LIN {X 0,Y 573.283,Z 236.698,A -85,B 0,C 180,E1 -2312.234,E2 -2312.234} C_VEL
LIN {X 0,Y 573.268,Z 236.699,A -85,B 0,C 180,E1 -2315.365,E2 -2315.365} C_VEL
LIN {X 0,Y 573.222,Z 236.703,A -85,B 0,C 180,E1 -2318.418,E2 -2318.418} C_VEL
LIN {X 0,Y 573.27,Z 236.695,A -85,B 0,C 180,E1 -2320.727,E2 -2320.727} C_VEL
LIN {X 0,Y 573.253,Z 236.706,A -85,B 0,C 180,E1 -2323.621,E2 -2323.621} C_VEL
LIN {X 0,Y 573.232,Z 236.7,A -85,B 0,C 180,E1 -2326.529,E2 -2326.529} C_VEL
LIN {X 0,Y 573.274,Z 236.694,A -85,B 0,C 180,E1 -2328.733,E2 -2328.733} C_VEL
LIN {X 0,Y 573.298,Z 236.7,A -85,B 0,C 180,E1 -2331.54,E2 -2331.54} C_VEL
LIN {X 0,Y 573.285,Z 236.694,A -85,B 0,C 180,E1 -2334.371,E2 -2334.371} C_VEL
LIN {X 0,Y 573.304,Z 236.698,A -85,B 0,C 180,E1 -2337.188,E2 -2337.188} C_VEL
LIN {X 0,Y 573.307,Z 236.691,A -85,B 0,C 180,E1 -2339.999,E2 -2339.999} C_VEL
LIN {X 0,Y 573.305,Z 236.694,A -85,B 0,C 180,E1 -2342.81,E2 -2342.81} C_VEL
LIN {X 0,Y 573.282,Z 236.696,A -85,B 0,C 180,E1 -2345.627,E2 -2345.627} C_VEL
LIN {X 0,Y 573.279,Z 236.696,A -85,B 0,C 180,E1 -2348.458,E2 -2348.458} C_VEL
LIN {X 0,Y 573.287,Z 236.699,A -85,B 0,C 180,E1 -2351.311,E2 -2351.311} C_VEL
LIN {X 0,Y 573.268,Z 236.697,A -85,B 0,C 180,E1 -2354.424,E2 -2354.424} C_VEL
LIN {X 0,Y 573.246,Z 236.705,A -85,B 0,C 180,E1 -2357.111,E2 -2357.111} C_VEL
LIN {X 0,Y 573.245,Z 236.699,A -85,B 0,C 180,E1 -2360.076,E2 -2360.076} C_VEL
LIN {X 0,Y 573.258,Z 236.7,A -85,B 0,C 180,E1 -2363.153,E2 -2363.153} C_VEL
LIN {X 0,Y 573.241,Z 236.703,A -85,B 0,C 180,E1 -2364.403,E2 -2364.403} C_VEL
LIN {X 0,Y 572.608,Z 236.788,A -85,B 0,C 180,E1 -2364.99,E2 -2364.99} C_VEL
LIN {X 0,Y 569.762,Z 237.142,A -85,B 0,C 180,E1 -2365.941,E2 -2365.941} C_VEL
LIN {X 0,Y 567.334,Z 237.444,A -85,B 0,C 180,E1 -2366.707,E2 -2366.707} C_VEL
LIN {X 0,Y 566.285,Z 237.568,A -85,B 0,C 180,E1 -2367.298,E2 -2367.298} C_VEL
LIN {X 0,Y 566.197,Z 237.577,A -85,B 0,C 180,E1 -2367.498,E2 -2367.498} C_VEL
LIN {X 0,Y 566.212,Z 237.574,A -85,B 0,C 180,E1 -2369.767,E2 -2369.767} C_VEL
LIN {X 0,Y 566.191,Z 237.584,A -85,B 0,C 180,E1 -2372.43,E2 -2372.43} C_VEL
LIN {X 0,Y 566.188,Z 237.579,A -85,B 0,C 180,E1 -2374.992,E2 -2374.992} C_VEL
LIN {X 0,Y 566.181,Z 237.579,A -85,B 0,C 180,E1 -2377.46,E2 -2377.46} C_VEL
LIN {X 0,Y 566.212,Z 237.581,A -85,B 0,C 180,E1 -2380.197,E2 -2380.197} C_VEL
LIN {X 0,Y 566.196,Z 237.578,A -85,B 0,C 180,E1 -2383.053,E2 -2383.053} C_VEL
LIN {X 0,Y 566.186,Z 237.585,A -85,B 0,C 180,E1 -2386.048,E2 -2386.048} C_VEL
LIN {X 0,Y 566.196,Z 237.579,A -85,B 0,C 180,E1 -2388.864,E2 -2388.864} C_VEL
LIN {X 0,Y 566.175,Z 237.584,A -85,B 0,C 180,E1 -2391.637,E2 -2391.637} C_VEL
LIN {X 0,Y 566.214,Z 237.686,A -85,B 0,C 180,E1 -2394.485,E2 -2394.485} C_VEL
LIN {X 0,Y 566.846,Z 243.491,A -85,B 0,C 180,E1 -2395.444,E2 -2395.444} C_VEL
LIN {X 0,Y 566.584,Z 259.614,A -85,B 0,C 180,E1 -2397.977,E2 -2397.977} C_VEL
LIN {X 0,Y 566.546,Z 266.895,A -85,B 0,C 180,E1 -2399.084,E2 -2399.084} C_VEL
LIN {X 0,Y 567.77,Z 274.286,A -85,B 0,C 180,E1 -2399.217,E2 -2399.217} C_VEL
LIN {X 0,Y 567.426,Z 403.279,A -85,B 0,C 180,E1 -2400.888,E2 -2400.888} C_VEL
LIN {X 0,Y 567.276,Z 417.794,A -85,B 0,C 180,E1 -2401.223,E2 -2401.223} C_VEL
LIN {X 0,Y 567.143,Z 431.004,A -85,B 0,C 180,E1 -2401.667,E2 -2401.667} C_VEL
LIN {X 0,Y 566.989,Z 443.123,A -85,B 0,C 180,E1 -2402.202,E2 -2402.202} C_VEL
LIN {X 0,Y 566.761,Z 456.118,A -85,B 0,C 180,E1 -2402.929,E2 -2402.929} C_VEL
LIN {X 0,Y 566.557,Z 468.236,A -85,B 0,C 180,E1 -2403.774,E2 -2403.774} C_VEL
LIN {X 0,Y 566.389,Z 479.468,A -85,B 0,C 180,E1 -2404.731,E2 -2404.731} C_VEL
LIN {X 0,Y 566.253,Z 490.014,A -85,B 0,C 180,E1 -2405.822,E2 -2405.822} C_VEL
LIN {X 0,Y 566.139,Z 499.355,A -85,B 0,C 180,E1 -2406.999,E2 -2406.999} C_VEL
LIN {X 0,Y 566.041,Z 506.752,A -85,B 0,C 180,E1 -2408.132,E2 -2408.132} C_VEL
LIN {X 0,Y 565.961,Z 512.883,A -85,B 0,C 180,E1 -2409.274,E2 -2409.274} C_VEL
LIN {X 0,Y 565.955,Z 518.916,A -85,B 0,C 180,E1 -2410.688,E2 -2410.688} C_VEL
LIN {X 0,Y 565.898,Z 522.863,A -85,B 0,C 180,E1 -2411.912,E2 -2411.912} C_VEL
LIN {X 0,Y 565.861,Z 526.209,A -85,B 0,C 180,E1 -2413.402,E2 -2413.402} C_VEL
LIN {X 0,Y 565.827,Z 528.034,A -85,B 0,C 180,E1 -2414.881,E2 -2414.881} C_VEL
LIN {X 0,Y 565.854,Z 528.439,A -85,B 0,C 180,E1 -2416.351,E2 -2416.351} C_VEL
LIN {X 0,Y 565.859,Z 527.454,A -85,B 0,C 180,E1 -2417.811,E2 -2417.811} C_VEL
LIN {X 0,Y 565.879,Z 525.08,A -85,B 0,C 180,E1 -2419.264,E2 -2419.264} C_VEL
LIN {X 0,Y 565.878,Z 521.281,A -85,B 0,C 180,E1 -2420.709,E2 -2420.709} C_VEL
LIN {X 0,Y 565.952,Z 517.395,A -85,B 0,C 180,E1 -2421.79,E2 -2421.79} C_VEL
LIN {X 0,Y 565.985,Z 511.373,A -85,B 0,C 180,E1 -2423.115,E2 -2423.115} C_VEL
LIN {X 0,Y 566.037,Z 504.637,A -85,B 0,C 180,E1 -2424.3,E2 -2424.3} C_VEL
LIN {X 0,Y 566.174,Z 495.909,A -85,B 0,C 180,E1 -2425.551,E2 -2425.551} C_VEL
LIN {X 0,Y 566.285,Z 486.831,A -85,B 0,C 180,E1 -2426.621,E2 -2426.621} C_VEL
LIN {X 0,Y 566.438,Z 477.817,A -85,B 0,C 180,E1 -2427.511,E2 -2427.511} C_VEL
LIN {X 0,Y 566.611,Z 465.974,A -85,B 0,C 180,E1 -2428.49,E2 -2428.49} C_VEL
LIN {X 0,Y 566.825,Z 454.056,A -85,B 0,C 180,E1 -2429.29,E2 -2429.29} C_VEL
LIN {X 0,Y 567.036,Z 440.812,A -85,B 0,C 180,E1 -2430,E2 -2430} C_VEL
LIN {X 0,Y 567.188,Z 426.85,A -85,B 0,C 180,E1 -2430.577,E2 -2430.577} C_VEL
LIN {X 0,Y 567.32,Z 412.804,A -85,B 0,C 180,E1 -2430.998,E2 -2430.998} C_VEL
LIN {X 0,Y 567.413,Z 399.298,A -85,B 0,C 180,E1 -2431.264,E2 -2431.264} C_VEL
LIN {X 0,Y 567.674,Z 272.851,A -85,B 0,C 180,E1 -2432.894,E2 -2432.894} C_VEL
LIN {X 0,Y 566.499,Z 266.67,A -85,B 0,C 180,E1 -2433.022,E2 -2433.022} C_VEL
LIN {X 0,Y 566.729,Z 250.62,A -85,B 0,C 180,E1 -2435.515,E2 -2435.515} C_VEL
LIN {X 0,Y 566.793,Z 240.515,A -85,B 0,C 180,E1 -2437.123,E2 -2437.123} C_VEL
LIN {X 0,Y 566.242,Z 237.58,A -85,B 0,C 180,E1 -2437.65,E2 -2437.65} C_VEL
LIN {X 0,Y 566.238,Z 237.573,A -85,B 0,C 180,E1 -2440.73,E2 -2440.73} C_VEL
LIN {X 0,Y 566.194,Z 237.584,A -85,B 0,C 180,E1 -2443.641,E2 -2443.641} C_VEL
LIN {X 0,Y 566.21,Z 237.575,A -85,B 0,C 180,E1 -2446.588,E2 -2446.588} C_VEL
LIN {X 0,Y 566.201,Z 237.582,A -85,B 0,C 180,E1 -2449.581,E2 -2449.581} C_VEL
LIN {X 0,Y 566.184,Z 237.586,A -85,B 0,C 180,E1 -2451.863,E2 -2451.863} C_VEL
LIN {X 0,Y 566.22,Z 237.575,A -85,B 0,C 180,E1 -2455.034,E2 -2455.034} C_VEL
LIN {X 0,Y 566.214,Z 237.579,A -85,B 0,C 180,E1 -2457.338,E2 -2457.338} C_VEL
LIN {X 0,Y 566.214,Z 237.581,A -85,B 0,C 180,E1 -2459.767,E2 -2459.767} C_VEL
LIN {X 0,Y 566.198,Z 237.576,A -85,B 0,C 180,E1 -2462.432,E2 -2462.432} C_VEL
LIN {X 0,Y 566.201,Z 237.578,A -85,B 0,C 180,E1 -2464.995,E2 -2464.995} C_VEL
LIN {X 0,Y 566.183,Z 237.588,A -85,B 0,C 180,E1 -2467.461,E2 -2467.461} C_VEL
LIN {X 0,Y 566.213,Z 237.575,A -85,B 0,C 180,E1 -2470.198,E2 -2470.198} C_VEL
LIN {X 0,Y 566.198,Z 237.581,A -85,B 0,C 180,E1 -2473.053,E2 -2473.053} C_VEL
LIN {X 0,Y 566.188,Z 237.578,A -85,B 0,C 180,E1 -2476.049,E2 -2476.049} C_VEL
LIN {X 0,Y 566.207,Z 237.579,A -85,B 0,C 180,E1 -2478.865,E2 -2478.865} C_VEL
LIN {X 0,Y 566.179,Z 237.582,A -85,B 0,C 180,E1 -2481.638,E2 -2481.638} C_VEL
LIN {X 0,Y 566.2,Z 237.576,A -85,B 0,C 180,E1 -2484.312,E2 -2484.312} C_VEL
LIN {X 0,Y 566.215,Z 237.581,A -85,B 0,C 180,E1 -2486.899,E2 -2486.899} C_VEL
LIN {X 0,Y 566.182,Z 237.582,A -85,B 0,C 180,E1 -2489.409,E2 -2489.409} C_VEL
LIN {X 0,Y 566.215,Z 237.574,A -85,B 0,C 180,E1 -2491.859,E2 -2491.859} C_VEL
LIN {X 0,Y 566.214,Z 237.575,A -85,B 0,C 180,E1 -2494.252,E2 -2494.252} C_VEL
LIN {X 0,Y 566.181,Z 237.585,A -85,B 0,C 180,E1 -2496.714,E2 -2496.714} C_VEL
LIN {X 0,Y 566.209,Z 237.575,A -85,B 0,C 180,E1 -2499.664,E2 -2499.664} C_VEL
LIN {X 0,Y 566.194,Z 237.584,A -85,B 0,C 180,E1 -2502.669,E2 -2502.669} C_VEL
LIN {X 0,Y 566.223,Z 237.573,A -85,B 0,C 180,E1 -2505.628,E2 -2505.628} C_VEL
LIN {X 0,Y 566.223,Z 237.583,A -85,B 0,C 180,E1 -2508.676,E2 -2508.676} C_VEL
LIN {X 0,Y 566.226,Z 237.573,A -85,B 0,C 180,E1 -2511.435,E2 -2511.435} C_VEL
LIN {X 0,Y 566.253,Z 237.575,A -85,B 0,C 180,E1 -2514.303,E2 -2514.303} C_VEL
LIN {X 0,Y 566.272,Z 237.568,A -85,B 0,C 180,E1 -2517.867,E2 -2517.867} C_VEL
LIN {X 0,Y 566.298,Z 237.57,A -85,B 0,C 180,E1 -2520.712,E2 -2520.712} C_VEL
LIN {X 0,Y 566.269,Z 237.571,A -85,B 0,C 180,E1 -2522.846,E2 -2522.846} C_VEL
LIN {X 0,Y 566.254,Z 237.57,A -85,B 0,C 180,E1 -2525.699,E2 -2525.699} C_VEL
LIN {X 0,Y 566.227,Z 237.579,A -85,B 0,C 180,E1 -2528.567,E2 -2528.567} C_VEL
LIN {X 0,Y 566.234,Z 237.572,A -85,B 0,C 180,E1 -2531.455,E2 -2531.455} C_VEL
LIN {X 0,Y 566.227,Z 237.578,A -85,B 0,C 180,E1 -2534.508,E2 -2534.508} C_VEL
LIN {X 0,Y 566.198,Z 237.577,A -85,B 0,C 180,E1 -2537.332,E2 -2537.332} C_VEL
LIN {X 0,Y 566.209,Z 237.581,A -85,B 0,C 180,E1 -2540.338,E2 -2540.338} C_VEL
LIN {X 0,Y 566.185,Z 237.579,A -85,B 0,C 180,E1 -2543.405,E2 -2543.405} C_VEL
LIN {X 0,Y 566.209,Z 237.58,A -85,B 0,C 180,E1 -2545.75,E2 -2545.75} C_VEL
LIN {X 0,Y 566.201,Z 237.582,A -85,B 0,C 180,E1 -2548.204,E2 -2548.204} C_VEL
LIN {X 0,Y 566.189,Z 237.578,A -85,B 0,C 180,E1 -2550.593,E2 -2550.593} C_VEL
LIN {X 0,Y 566.225,Z 237.573,A -85,B 0,C 180,E1 -2553.103,E2 -2553.103} C_VEL
LIN {X 0,Y 566.209,Z 237.582,A -85,B 0,C 180,E1 -2555.689,E2 -2555.689} C_VEL
LIN {X 0,Y 566.213,Z 237.575,A -85,B 0,C 180,E1 -2558.56,E2 -2558.56} C_VEL
LIN {X 0,Y 566.201,Z 237.578,A -85,B 0,C 180,E1 -2561.138,E2 -2561.138} C_VEL
LIN {X 0,Y 566.195,Z 237.581,A -85,B 0,C 180,E1 -2564.037,E2 -2564.037} C_VEL
LIN {X 0,Y 566.204,Z 237.578,A -85,B 0,C 180,E1 -2567.083,E2 -2567.083} C_VEL
LIN {X 0,Y 566.205,Z 237.582,A -85,B 0,C 180,E1 -2569.802,E2 -2569.802} C_VEL
LIN {X 0,Y 566.197,Z 237.576,A -85,B 0,C 180,E1 -2572.6,E2 -2572.6} C_VEL
LIN {X 0,Y 566.199,Z 237.581,A -85,B 0,C 180,E1 -2575.182,E2 -2575.182} C_VEL
LIN {X 0,Y 566.233,Z 237.579,A -85,B 0,C 180,E1 -2577.744,E2 -2577.744} C_VEL
LIN {X 0,Y 566.203,Z 237.577,A -85,B 0,C 180,E1 -2580.329,E2 -2580.329} C_VEL
LIN {X 0,Y 566.212,Z 237.578,A -85,B 0,C 180,E1 -2582.662,E2 -2582.662} C_VEL
LIN {X 0,Y 566.263,Z 237.689,A -85,B 0,C 180,E1 -2585.261,E2 -2585.261} C_VEL
LIN {X 0,Y 567.317,Z 243.08,A -85,B 0,C 180,E1 -2586.044,E2 -2586.044} C_VEL
LIN {X 0,Y 567.119,Z 262.492,A -85,B 0,C 180,E1 -2588.647,E2 -2588.647} C_VEL
LIN {X 0,Y 566.829,Z 284.536,A -85,B 0,C 180,E1 -2591.569,E2 -2591.569} C_VEL
LIN {X 0,Y 566.669,Z 295.557,A -85,B 0,C 180,E1 -2593.018,E2 -2593.018} C_VEL
LIN {X 0,Y 567.791,Z 302.851,A -85,B 0,C 180,E1 -2593.155,E2 -2593.155} C_VEL
LIN {X 0,Y 567.434,Z 433.897,A -85,B 0,C 180,E1 -2594.856,E2 -2594.856} C_VEL
LIN {X 0,Y 567.268,Z 448.613,A -85,B 0,C 180,E1 -2595.202,E2 -2595.202} C_VEL
LIN {X 0,Y 567.112,Z 462.843,A -85,B 0,C 180,E1 -2595.696,E2 -2595.696} C_VEL
LIN {X 0,Y 566.963,Z 475.645,A -85,B 0,C 180,E1 -2596.286,E2 -2596.286} C_VEL
LIN {X 0,Y 566.755,Z 488.106,A -85,B 0,C 180,E1 -2597.012,E2 -2597.012} C_VEL
LIN {X 0,Y 566.572,Z 500.647,A -85,B 0,C 180,E1 -2597.917,E2 -2597.917} C_VEL
LIN {X 0,Y 566.447,Z 511.321,A -85,B 0,C 180,E1 -2598.861,E2 -2598.861} C_VEL
LIN {X 0,Y 566.206,Z 521.853,A -85,B 0,C 180,E1 -2599.993,E2 -2599.993} C_VEL
LIN {X 0,Y 566.137,Z 530.174,A -85,B 0,C 180,E1 -2601.073,E2 -2601.073} C_VEL
LIN {X 0,Y 566.047,Z 538.128,A -85,B 0,C 180,E1 -2602.33,E2 -2602.33} C_VEL
LIN {X 0,Y 565.945,Z 544.528,A -85,B 0,C 180,E1 -2603.583,E2 -2603.583} C_VEL
LIN {X 0,Y 565.928,Z 548.961,A -85,B 0,C 180,E1 -2604.656,E2 -2604.656} C_VEL
LIN {X 0,Y 565.956,Z 552.443,A -85,B 0,C 180,E1 -2605.727,E2 -2605.727} C_VEL
LIN {X 0,Y 565.875,Z 555.832,A -85,B 0,C 180,E1 -2607.152,E2 -2607.152} C_VEL
LIN {X 0,Y 565.841,Z 557.833,A -85,B 0,C 180,E1 -2608.577,E2 -2608.577} C_VEL
LIN {X 0,Y 565.837,Z 558.5,A -85,B 0,C 180,E1 -2610,E2 -2610} C_VEL
LIN {X 0,Y 565.841,Z 557.834,A -85,B 0,C 180,E1 -2611.423,E2 -2611.423} C_VEL
LIN {X 0,Y 565.875,Z 555.835,A -85,B 0,C 180,E1 -2612.847,E2 -2612.847} C_VEL
LIN {X 0,Y 565.956,Z 552.446,A -85,B 0,C 180,E1 -2614.273,E2 -2614.273} C_VEL
LIN {X 0,Y 565.985,Z 547.569,A -85,B 0,C 180,E1 -2615.701,E2 -2615.701} C_VEL
LIN {X 0,Y 565.996,Z 543.045,A -85,B 0,C 180,E1 -2616.738,E2 -2616.738} C_VEL
LIN {X 0,Y 566.047,Z 536.038,A -85,B 0,C 180,E1 -2618.029,E2 -2618.029} C_VEL
LIN {X 0,Y 566.177,Z 527.56,A -85,B 0,C 180,E1 -2619.286,E2 -2619.286} C_VEL
LIN {X 0,Y 566.294,Z 518.71,A -85,B 0,C 180,E1 -2620.367,E2 -2620.367} C_VEL
LIN {X 0,Y 566.467,Z 507.992,A -85,B 0,C 180,E1 -2621.449,E2 -2621.449} C_VEL
LIN {X 0,Y 566.611,Z 497.143,A -85,B 0,C 180,E1 -2622.354,E2 -2622.354} C_VEL
LIN {X 0,Y 566.79,Z 485.26,A -85,B 0,C 180,E1 -2623.17,E2 -2623.17} C_VEL
LIN {X 0,Y 567.035,Z 472.104,A -85,B 0,C 180,E1 -2623.894,E2 -2623.894} C_VEL
LIN {X 0,Y 567.235,Z 459.039,A -85,B 0,C 180,E1 -2624.453,E2 -2624.453} C_VEL
LIN {X 0,Y 567.354,Z 445.151,A -85,B 0,C 180,E1 -2624.893,E2 -2624.893} C_VEL
LIN {X 0,Y 567.428,Z 431.157,A -85,B 0,C 180,E1 -2625.19,E2 -2625.19} C_VEL
LIN {X 0,Y 567.737,Z 301.687,A -85,B 0,C 180,E1 -2626.862,E2 -2626.862} C_VEL
LIN {X 0,Y 566.666,Z 295.559,A -85,B 0,C 180,E1 -2626.982,E2 -2626.982} C_VEL
LIN {X 0,Y 566.964,Z 274.789,A -85,B 0,C 180,E1 -2629.722,E2 -2629.722} C_VEL
LIN {X 0,Y 567.271,Z 253.229,A -85,B 0,C 180,E1 -2632.585,E2 -2632.585} C_VEL
LIN {X 0,Y 567.297,Z 243.048,A -85,B 0,C 180,E1 -2633.958,E2 -2633.958} C_VEL
LIN {X 0,Y 566.256,Z 237.58,A -85,B 0,C 180,E1 -2634.763,E2 -2634.763} C_VEL
LIN {X 0,Y 566.211,Z 237.577,A -85,B 0,C 180,E1 -2637.338,E2 -2637.338} C_VEL
LIN {X 0,Y 566.201,Z 237.578,A -85,B 0,C 180,E1 -2639.768,E2 -2639.768} C_VEL
LIN {X 0,Y 566.206,Z 237.585,A -85,B 0,C 180,E1 -2642.43,E2 -2642.43} C_VEL
LIN {X 0,Y 566.18,Z 237.583,A -85,B 0,C 180,E1 -2644.989,E2 -2644.989} C_VEL
LIN {X 0,Y 566.194,Z 237.577,A -85,B 0,C 180,E1 -2647.46,E2 -2647.46} C_VEL
LIN {X 0,Y 566.204,Z 237.584,A -85,B 0,C 180,E1 -2650.198,E2 -2650.198} C_VEL
LIN {X 0,Y 566.203,Z 237.577,A -85,B 0,C 180,E1 -2653.053,E2 -2653.053} C_VEL
LIN {X 0,Y 566.195,Z 237.584,A -85,B 0,C 180,E1 -2656.048,E2 -2656.048} C_VEL
LIN {X 0,Y 566.208,Z 237.577,A -85,B 0,C 180,E1 -2658.863,E2 -2658.863} C_VEL
LIN {X 0,Y 566.186,Z 237.581,A -85,B 0,C 180,E1 -2661.636,E2 -2661.636} C_VEL
LIN {X 0,Y 566.208,Z 237.578,A -85,B 0,C 180,E1 -2664.311,E2 -2664.311} C_VEL
LIN {X 0,Y 566.224,Z 237.574,A -85,B 0,C 180,E1 -2666.897,E2 -2666.897} C_VEL
LIN {X 0,Y 566.188,Z 237.579,A -85,B 0,C 180,E1 -2669.407,E2 -2669.407} C_VEL
LIN {X 0,Y 566.222,Z 237.582,A -85,B 0,C 180,E1 -2671.857,E2 -2671.857} C_VEL
LIN {X 0,Y 566.208,Z 237.579,A -85,B 0,C 180,E1 -2674.25,E2 -2674.25} C_VEL
LIN {X 0,Y 566.185,Z 237.578,A -85,B 0,C 180,E1 -2676.713,E2 -2676.713} C_VEL
LIN {X 0,Y 566.208,Z 237.584,A -85,B 0,C 180,E1 -2679.662,E2 -2679.662} C_VEL
LIN {X 0,Y 566.197,Z 237.577,A -85,B 0,C 180,E1 -2682.668,E2 -2682.668} C_VEL
LIN {X 0,Y 566.226,Z 237.583,A -85,B 0,C 180,E1 -2685.626,E2 -2685.626} C_VEL
LIN {X 0,Y 566.267,Z 237.567,A -85,B 0,C 180,E1 -2688.653,E2 -2688.653} C_VEL
LIN {X 0,Y 566.24,Z 237.581,A -85,B 0,C 180,E1 -2691.434,E2 -2691.434} C_VEL
LIN {X 0,Y 566.252,Z 237.57,A -85,B 0,C 180,E1 -2694.301,E2 -2694.301} C_VEL
LIN {X 0,Y 566.27,Z 237.574,A -85,B 0,C 180,E1 -2697.154,E2 -2697.154} C_VEL
LIN {X 0,Y 566.277,Z 237.567,A -85,B 0,C 180,E1 -2699.999,E2 -2699.999} C_VEL
LIN {X 0,Y 566.27,Z 237.571,A -85,B 0,C 180,E1 -2702.845,E2 -2702.845} C_VEL
LIN {X 0,Y 566.25,Z 237.571,A -85,B 0,C 180,E1 -2705.697,E2 -2705.697} C_VEL
LIN {X 0,Y 566.223,Z 237.576,A -85,B 0,C 180,E1 -2708.565,E2 -2708.565} C_VEL
LIN {X 0,Y 566.239,Z 237.575,A -85,B 0,C 180,E1 -2711.453,E2 -2711.453} C_VEL
LIN {X 0,Y 566.221,Z 237.576,A -85,B 0,C 180,E1 -2714.506,E2 -2714.506} C_VEL
LIN {X 0,Y 566.188,Z 237.581,A -85,B 0,C 180,E1 -2717.331,E2 -2717.331} C_VEL
LIN {X 0,Y 566.208,Z 237.578,A -85,B 0,C 180,E1 -2720.336,E2 -2720.336} C_VEL
LIN {X 0,Y 566.217,Z 237.575,A -85,B 0,C 180,E1 -2723.401,E2 -2723.401} C_VEL
LIN {X 0,Y 566.199,Z 237.577,A -85,B 0,C 180,E1 -2725.748,E2 -2725.748} C_VEL
LIN {X 0,Y 566.197,Z 237.577,A -85,B 0,C 180,E1 -2727.498,E2 -2727.498} C_VEL
LIN {X 0,Y 565.523,Z 237.664,A -85,B 0,C 180,E1 -2728.092,E2 -2728.092} C_VEL
LIN {X 0,Y 562.659,Z 238.02,A -85,B 0,C 180,E1 -2729.055,E2 -2729.055} C_VEL
LIN {X 0,Y 560.246,Z 238.32,A -85,B 0,C 180,E1 -2729.831,E2 -2729.831} C_VEL
LIN {X 0,Y 559.214,Z 238.452,A -85,B 0,C 180,E1 -2730.43,E2 -2730.43} C_VEL
LIN {X 0,Y 559.133,Z 238.457,A -85,B 0,C 180,E1 -2730.633,E2 -2730.633} C_VEL
LIN {X 0,Y 559.149,Z 238.455,A -85,B 0,C 180,E1 -2733.574,E2 -2733.574} C_VEL
LIN {X 0,Y 559.152,Z 238.462,A -85,B 0,C 180,E1 -2736.448,E2 -2736.448} C_VEL
LIN {X 0,Y 559.163,Z 238.455,A -85,B 0,C 180,E1 -2738.933,E2 -2738.933} C_VEL
LIN {X 0,Y 559.18,Z 238.453,A -85,B 0,C 180,E1 -2741.767,E2 -2741.767} C_VEL
LIN {X 0,Y 559.124,Z 238.462,A -85,B 0,C 180,E1 -2744.739,E2 -2744.739} C_VEL
LIN {X 0,Y 559.148,Z 238.456,A -85,B 0,C 180,E1 -2747.257,E2 -2747.257} C_VEL
LIN {X 0,Y 559.171,Z 238.462,A -85,B 0,C 180,E1 -2750.135,E2 -2750.135} C_VEL
LIN {X 0,Y 559.13,Z 238.462,A -85,B 0,C 180,E1 -2752.892,E2 -2752.892} C_VEL
LIN {X 0,Y 559.207,Z 238.602,A -85,B 0,C 180,E1 -2754.323,E2 -2754.323} C_VEL
LIN {X 0,Y 559.951,Z 243.649,A -85,B 0,C 180,E1 -2755.176,E2 -2755.176} C_VEL
LIN {X 0,Y 559.606,Z 261.03,A -85,B 0,C 180,E1 -2757.954,E2 -2757.954} C_VEL
LIN {X 0,Y 559.567,Z 266.769,A -85,B 0,C 180,E1 -2758.864,E2 -2758.864} C_VEL
LIN {X 0,Y 560.963,Z 274.225,A -85,B 0,C 180,E1 -2759.006,E2 -2759.006} C_VEL
LIN {X 0,Y 560.582,Z 403.558,A -85,B 0,C 180,E1 -2760.704,E2 -2760.704} C_VEL
LIN {X 0,Y 560.409,Z 417.899,A -85,B 0,C 180,E1 -2761.04,E2 -2761.04} C_VEL
LIN {X 0,Y 560.236,Z 432.09,A -85,B 0,C 180,E1 -2761.531,E2 -2761.531} C_VEL
LIN {X 0,Y 560.033,Z 445.125,A -85,B 0,C 180,E1 -2762.131,E2 -2762.131} C_VEL
LIN {X 0,Y 559.806,Z 457.281,A -85,B 0,C 180,E1 -2762.839,E2 -2762.839} C_VEL
LIN {X 0,Y 559.566,Z 469.557,A -85,B 0,C 180,E1 -2763.723,E2 -2763.723} C_VEL
LIN {X 0,Y 559.384,Z 480.79,A -85,B 0,C 180,E1 -2764.713,E2 -2764.713} C_VEL
LIN {X 0,Y 559.214,Z 490.045,A -85,B 0,C 180,E1 -2765.696,E2 -2765.696} C_VEL
LIN {X 0,Y 559.105,Z 498.891,A -85,B 0,C 180,E1 -2766.82,E2 -2766.82} C_VEL
LIN {X 0,Y 558.963,Z 506.712,A -85,B 0,C 180,E1 -2768.024,E2 -2768.024} C_VEL
LIN {X 0,Y 558.906,Z 511.946,A -85,B 0,C 180,E1 -2769,E2 -2769} C_VEL
LIN {X 0,Y 558.865,Z 517.099,A -85,B 0,C 180,E1 -2770.152,E2 -2770.152} C_VEL
LIN {X 0,Y 558.806,Z 521.202,A -85,B 0,C 180,E1 -2771.295,E2 -2771.295} C_VEL
LIN {X 0,Y 558.781,Z 525.335,A -85,B 0,C 180,E1 -2772.911,E2 -2772.911} C_VEL
LIN {X 0,Y 558.741,Z 527.084,A -85,B 0,C 180,E1 -2773.936,E2 -2773.936} C_VEL
LIN {X 0,Y 558.769,Z 528.371,A -85,B 0,C 180,E1 -2775.431,E2 -2775.431} C_VEL
LIN {X 0,Y 558.736,Z 528.238,A -85,B 0,C 180,E1 -2776.915,E2 -2776.915} C_VEL
LIN {X 0,Y 558.759,Z 526.721,A -85,B 0,C 180,E1 -2778.391,E2 -2778.391} C_VEL
LIN {X 0,Y 558.79,Z 523.803,A -85,B 0,C 180,E1 -2779.859,E2 -2779.859} C_VEL
LIN {X 0,Y 558.824,Z 519.431,A -85,B 0,C 180,E1 -2781.32,E2 -2781.32} C_VEL
LIN {X 0,Y 558.892,Z 515.108,A -85,B 0,C 180,E1 -2782.413,E2 -2782.413} C_VEL
LIN {X 0,Y 558.962,Z 508.843,A -85,B 0,C 180,E1 -2783.684,E2 -2783.684} C_VEL
LIN {X 0,Y 559.054,Z 501.081,A -85,B 0,C 180,E1 -2784.952,E2 -2784.952} C_VEL
LIN {X 0,Y 559.138,Z 493.023,A -85,B 0,C 180,E1 -2786.036,E2 -2786.036} C_VEL
LIN {X 0,Y 559.363,Z 483.341,A -85,B 0,C 180,E1 -2787.119,E2 -2787.119} C_VEL
LIN {X 0,Y 559.538,Z 471.623,A -85,B 0,C 180,E1 -2788.201,E2 -2788.201} C_VEL
LIN {X 0,Y 559.775,Z 459.598,A -85,B 0,C 180,E1 -2789.101,E2 -2789.101} C_VEL
LIN {X 0,Y 560.006,Z 447.769,A -85,B 0,C 180,E1 -2789.82,E2 -2789.82} C_VEL
LIN {X 0,Y 560.221,Z 433.691,A -85,B 0,C 180,E1 -2790.494,E2 -2790.494} C_VEL
LIN {X 0,Y 560.396,Z 419.2,A -85,B 0,C 180,E1 -2791.011,E2 -2791.011} C_VEL
LIN {X 0,Y 560.5,Z 405.571,A -85,B 0,C 180,E1 -2791.347,E2 -2791.347} C_VEL
LIN {X 0,Y 560.653,Z 380.313,A -85,B 0,C 180,E1 -2791.706,E2 -2791.706} C_VEL
LIN {X 0,Y 560.842,Z 273.439,A -85,B 0,C 180,E1 -2793.098,E2 -2793.098} C_VEL
LIN {X 0,Y 559.538,Z 266.685,A -85,B 0,C 180,E1 -2793.24,E2 -2793.24} C_VEL
LIN {X 0,Y 559.844,Z 248.533,A -85,B 0,C 180,E1 -2796.125,E2 -2796.125} C_VEL
LIN {X 0,Y 559.839,Z 241.817,A -85,B 0,C 180,E1 -2797.212,E2 -2797.212} C_VEL
LIN {X 0,Y 559.2,Z 238.458,A -85,B 0,C 180,E1 -2797.796,E2 -2797.796} C_VEL
LIN {X 0,Y 559.2,Z 238.45,A -85,B 0,C 180,E1 -2800.866,E2 -2800.866} C_VEL
LIN {X 0,Y 559.168,Z 238.461,A -85,B 0,C 180,E1 -2803.816,E2 -2803.816} C_VEL
LIN {X 0,Y 559.173,Z 238.451,A -85,B 0,C 180,E1 -2806.802,E2 -2806.802} C_VEL
LIN {X 0,Y 559.162,Z 238.462,A -85,B 0,C 180,E1 -2809.837,E2 -2809.837} C_VEL
LIN {X 0,Y 559.13,Z 238.46,A -85,B 0,C 180,E1 -2812.153,E2 -2812.153} C_VEL
LIN {X 0,Y 559.192,Z 238.452,A -85,B 0,C 180,E1 -2815.193,E2 -2815.193} C_VEL
LIN {X 0,Y 559.182,Z 238.459,A -85,B 0,C 180,E1 -2817.712,E2 -2817.712} C_VEL
LIN {X 0,Y 559.155,Z 238.455,A -85,B 0,C 180,E1 -2820.182,E2 -2820.182} C_VEL
LIN {X 0,Y 559.163,Z 238.453,A -85,B 0,C 180,E1 -2822.714,E2 -2822.714} C_VEL
LIN {X 0,Y 559.145,Z 238.462,A -85,B 0,C 180,E1 -2825.322,E2 -2825.322} C_VEL
LIN {X 0,Y 559.122,Z 238.46,A -85,B 0,C 180,E1 -2828.018,E2 -2828.018} C_VEL
LIN {X 0,Y 559.166,Z 238.454,A -85,B 0,C 180,E1 -2830.811,E2 -2830.811} C_VEL
LIN {X 0,Y 559.15,Z 238.458,A -85,B 0,C 180,E1 -2833.732,E2 -2833.732} C_VEL
LIN {X 0,Y 559.159,Z 238.456,A -85,B 0,C 180,E1 -2836.801,E2 -2836.801} C_VEL
LIN {X 0,Y 559.166,Z 238.462,A -85,B 0,C 180,E1 -2839.19,E2 -2839.19} C_VEL
LIN {X 0,Y 559.123,Z 238.458,A -85,B 0,C 180,E1 -2841.983,E2 -2841.983} C_VEL
LIN {X 0,Y 559.147,Z 238.458,A -85,B 0,C 180,E1 -2844.679,E2 -2844.679} C_VEL
LIN {X 0,Y 559.161,Z 238.458,A -85,B 0,C 180,E1 -2847.362,E2 -2847.362} C_VEL
LIN {X 0,Y 559.177,Z 238.451,A -85,B 0,C 180,E1 -2850.136,E2 -2850.136} C_VEL
LIN {X 0,Y 559.172,Z 238.458,A -85,B 0,C 180,E1 -2853.17,E2 -2853.17} C_VEL
LIN {X 0,Y 559.145,Z 238.457,A -85,B 0,C 180,E1 -2855.496,E2 -2855.496} C_VEL
LIN {X 0,Y 559.165,Z 238.458,A -85,B 0,C 180,E1 -2858.625,E2 -2858.625} C_VEL
LIN {X 0,Y 559.16,Z 238.461,A -85,B 0,C 180,E1 -2860.927,E2 -2860.927} C_VEL
LIN {X 0,Y 559.162,Z 238.453,A -85,B 0,C 180,E1 -2863.949,E2 -2863.949} C_VEL
LIN {X 0,Y 559.166,Z 238.454,A -85,B 0,C 180,E1 -2866.185,E2 -2866.185} C_VEL
LIN {X 0,Y 559.185,Z 238.453,A -85,B 0,C 180,E1 -2869.134,E2 -2869.134} C_VEL
LIN {X 0,Y 559.198,Z 238.45,A -85,B 0,C 180,E1 -2872.055,E2 -2872.055} C_VEL
LIN {X 0,Y 559.249,Z 238.446,A -85,B 0,C 180,E1 -2874.954,E2 -2874.954} C_VEL
LIN {X 0,Y 559.244,Z 238.444,A -85,B 0,C 180,E1 -2877.84,E2 -2877.84} C_VEL
LIN {X 0,Y 559.268,Z 238.445,A -85,B 0,C 180,E1 -2880.721,E2 -2880.721} C_VEL
LIN {X 0,Y 559.235,Z 238.447,A -85,B 0,C 180,E1 -2882.882,E2 -2882.882} C_VEL
LIN {X 0,Y 559.223,Z 238.447,A -85,B 0,C 180,E1 -2885.771,E2 -2885.771} C_VEL
LIN {X 0,Y 559.186,Z 238.454,A -85,B 0,C 180,E1 -2888.675,E2 -2888.675} C_VEL
LIN {X 0,Y 559.198,Z 238.449,A -85,B 0,C 180,E1 -2891.601,E2 -2891.601} C_VEL
LIN {X 0,Y 559.193,Z 238.453,A -85,B 0,C 180,E1 -2894.597,E2 -2894.597} C_VEL
LIN {X 0,Y 559.157,Z 238.455,A -85,B 0,C 180,E1 -2897.558,E2 -2897.558} C_VEL
LIN {X 0,Y 559.167,Z 238.457,A -85,B 0,C 180,E1 -2899.838,E2 -2899.838} C_VEL
LIN {X 0,Y 559.136,Z 238.465,A -85,B 0,C 180,E1 -2902.154,E2 -2902.154} C_VEL
LIN {X 0,Y 559.174,Z 238.451,A -85,B 0,C 180,E1 -2905.188,E2 -2905.188} C_VEL
LIN {X 0,Y 559.188,Z 238.455,A -85,B 0,C 180,E1 -2907.712,E2 -2907.712} C_VEL
LIN {X 0,Y 559.164,Z 238.458,A -85,B 0,C 180,E1 -2910.183,E2 -2910.183} C_VEL
LIN {X 0,Y 559.171,Z 238.452,A -85,B 0,C 180,E1 -2912.715,E2 -2912.715} C_VEL
LIN {X 0,Y 559.154,Z 238.456,A -85,B 0,C 180,E1 -2915.323,E2 -2915.323} C_VEL
LIN {X 0,Y 559.132,Z 238.463,A -85,B 0,C 180,E1 -2918.018,E2 -2918.018} C_VEL
LIN {X 0,Y 559.171,Z 238.452,A -85,B 0,C 180,E1 -2920.812,E2 -2920.812} C_VEL
LIN {X 0,Y 559.157,Z 238.463,A -85,B 0,C 180,E1 -2923.733,E2 -2923.733} C_VEL
LIN {X 0,Y 559.149,Z 238.455,A -85,B 0,C 180,E1 -2926.804,E2 -2926.804} C_VEL
LIN {X 0,Y 559.158,Z 238.457,A -85,B 0,C 180,E1 -2929.189,E2 -2929.189} C_VEL
LIN {X 0,Y 559.132,Z 238.46,A -85,B 0,C 180,E1 -2931.983,E2 -2931.983} C_VEL
LIN {X 0,Y 559.132,Z 238.457,A -85,B 0,C 180,E1 -2934.788,E2 -2934.788} C_VEL
LIN {X 0,Y 559.174,Z 238.46,A -85,B 0,C 180,E1 -2937.362,E2 -2937.362} C_VEL
LIN {X 0,Y 559.149,Z 238.457,A -85,B 0,C 180,E1 -2940.143,E2 -2940.143} C_VEL
LIN {X 0,Y 559.171,Z 238.46,A -85,B 0,C 180,E1 -2943.098,E2 -2943.098} C_VEL
LIN {X 0,Y 559.235,Z 238.613,A -85,B 0,C 180,E1 -2945.079,E2 -2945.079} C_VEL
LIN {X 0,Y 560.407,Z 244.507,A -85,B 0,C 180,E1 -2945.948,E2 -2945.948} C_VEL
LIN {X 0,Y 560.225,Z 260.881,A -85,B 0,C 180,E1 -2948.176,E2 -2948.176} C_VEL
LIN {X 0,Y 559.904,Z 283.06,A -85,B 0,C 180,E1 -2951.143,E2 -2951.143} C_VEL
LIN {X 0,Y 559.731,Z 295.547,A -85,B 0,C 180,E1 -2952.8,E2 -2952.8} C_VEL
LIN {X 0,Y 560.998,Z 303.112,A -85,B 0,C 180,E1 -2952.948,E2 -2952.948} C_VEL
LIN {X 0,Y 560.591,Z 433.897,A -85,B 0,C 180,E1 -2954.666,E2 -2954.666} C_VEL
LIN {X 0,Y 560.439,Z 448.467,A -85,B 0,C 180,E1 -2955.013,E2 -2955.013} C_VEL
LIN {X 0,Y 560.234,Z 462.841,A -85,B 0,C 180,E1 -2955.516,E2 -2955.516} C_VEL
LIN {X 0,Y 560.059,Z 475.643,A -85,B 0,C 180,E1 -2956.114,E2 -2956.114} C_VEL
LIN {X 0,Y 559.833,Z 488.104,A -85,B 0,C 180,E1 -2956.848,E2 -2956.848} C_VEL
LIN {X 0,Y 559.592,Z 500.649,A -85,B 0,C 180,E1 -2957.764,E2 -2957.764} C_VEL
LIN {X 0,Y 559.428,Z 511.74,A -85,B 0,C 180,E1 -2958.762,E2 -2958.762} C_VEL
LIN {X 0,Y 559.186,Z 521.854,A -85,B 0,C 180,E1 -2959.866,E2 -2959.866} C_VEL
LIN {X 0,Y 559.073,Z 530.175,A -85,B 0,C 180,E1 -2960.959,E2 -2960.959} C_VEL
LIN {X 0,Y 558.973,Z 538.128,A -85,B 0,C 180,E1 -2962.232,E2 -2962.232} C_VEL
LIN {X 0,Y 558.873,Z 544.528,A -85,B 0,C 180,E1 -2963.502,E2 -2963.502} C_VEL
LIN {X 0,Y 558.859,Z 548.961,A -85,B 0,C 180,E1 -2964.588,E2 -2964.588} C_VEL
LIN {X 0,Y 558.865,Z 552.444,A -85,B 0,C 180,E1 -2965.673,E2 -2965.673} C_VEL
LIN {X 0,Y 558.796,Z 555.832,A -85,B 0,C 180,E1 -2967.116,E2 -2967.116} C_VEL
LIN {X 0,Y 558.74,Z 557.834,A -85,B 0,C 180,E1 -2968.558,E2 -2968.558} C_VEL
LIN {X 0,Y 558.738,Z 558.5,A -85,B 0,C 180,E1 -2970,E2 -2970} C_VEL
LIN {X 0,Y 558.74,Z 557.835,A -85,B 0,C 180,E1 -2971.441,E2 -2971.441} C_VEL
LIN {X 0,Y 558.796,Z 555.835,A -85,B 0,C 180,E1 -2972.884,E2 -2972.884} C_VEL
LIN {X 0,Y 558.865,Z 552.447,A -85,B 0,C 180,E1 -2974.327,E2 -2974.327} C_VEL
LIN {X 0,Y 558.915,Z 547.569,A -85,B 0,C 180,E1 -2975.773,E2 -2975.773} C_VEL
LIN {X 0,Y 558.907,Z 541.055,A -85,B 0,C 180,E1 -2977.224,E2 -2977.224} C_VEL
LIN {X 0,Y 559.028,Z 533.804,A -85,B 0,C 180,E1 -2978.494,E2 -2978.494} C_VEL
LIN {X 0,Y 559.147,Z 524.824,A -85,B 0,C 180,E1 -2979.769,E2 -2979.769} C_VEL
LIN {X 0,Y 559.351,Z 515.396,A -85,B 0,C 180,E1 -2980.863,E2 -2980.863} C_VEL
LIN {X 0,Y 559.518,Z 504.958,A -85,B 0,C 180,E1 -2981.869,E2 -2981.869} C_VEL
LIN {X 0,Y 559.697,Z 493.436,A -85,B 0,C 180,E1 -2982.786,E2 -2982.786} C_VEL
LIN {X 0,Y 559.952,Z 480.647,A -85,B 0,C 180,E1 -2983.611,E2 -2983.611} C_VEL
LIN {X 0,Y 560.142,Z 468.156,A -85,B 0,C 180,E1 -2984.254,E2 -2984.254} C_VEL
LIN {X 0,Y 560.384,Z 455.088,A -85,B 0,C 180,E1 -2984.775,E2 -2984.775} C_VEL
LIN {X 0,Y 560.501,Z 441.608,A -85,B 0,C 180,E1 -2985.17,E2 -2985.17} C_VEL
LIN {X 0,Y 560.614,Z 426.632,A -85,B 0,C 180,E1 -2985.449,E2 -2985.449} C_VEL
LIN {X 0,Y 560.92,Z 302.267,A -85,B 0,C 180,E1 -2987.066,E2 -2987.066} C_VEL
LIN {X 0,Y 559.723,Z 295.605,A -85,B 0,C 180,E1 -2987.193,E2 -2987.193} C_VEL
LIN {X 0,Y 560.022,Z 274.487,A -85,B 0,C 180,E1 -2989.997,E2 -2989.997} C_VEL
LIN {X 0,Y 560.387,Z 251.611,A -85,B 0,C 180,E1 -2993.073,E2 -2993.073} C_VEL
LIN {X 0,Y 560.401,Z 244.475,A -85,B 0,C 180,E1 -2994.052,E2 -2994.052} C_VEL
LIN {X 0,Y 559.205,Z 238.457,A -85,B 0,C 180,E1 -2994.948,E2 -2994.948} C_VEL
LIN {X 0,Y 559.157,Z 238.455,A -85,B 0,C 180,E1 -2997.713,E2 -2997.713} C_VEL
LIN {X 0,Y 559.154,Z 238.459,A -85,B 0,C 180,E1 -3000.182,E2 -3000.182} C_VEL
LIN {X 0,Y 559.175,Z 238.461,A -85,B 0,C 180,E1 -3002.713,E2 -3002.713} C_VEL
LIN {X 0,Y 559.127,Z 238.46,A -85,B 0,C 180,E1 -3005.323,E2 -3005.323} C_VEL
LIN {X 0,Y 559.131,Z 238.461,A -85,B 0,C 180,E1 -3008.017,E2 -3008.017} C_VEL
LIN {X 0,Y 559.157,Z 238.456,A -85,B 0,C 180,E1 -3010.811,E2 -3010.811} C_VEL
LIN {X 0,Y 559.16,Z 238.456,A -85,B 0,C 180,E1 -3013.731,E2 -3013.731} C_VEL
LIN {X 0,Y 559.143,Z 238.457,A -85,B 0,C 180,E1 -3016.802,E2 -3016.802} C_VEL
LIN {X 0,Y 559.173,Z 238.452,A -85,B 0,C 180,E1 -3019.188,E2 -3019.188} C_VEL
LIN {X 0,Y 559.131,Z 238.465,A -85,B 0,C 180,E1 -3021.982,E2 -3021.982} C_VEL
LIN {X 0,Y 559.155,Z 238.452,A -85,B 0,C 180,E1 -3024.782,E2 -3024.782} C_VEL
LIN {X 0,Y 559.169,Z 238.454,A -85,B 0,C 180,E1 -3027.36,E2 -3027.36} C_VEL
LIN {X 0,Y 559.183,Z 238.457,A -85,B 0,C 180,E1 -3030.134,E2 -3030.134} C_VEL
LIN {X 0,Y 559.166,Z 238.453,A -85,B 0,C 180,E1 -3033.171,E2 -3033.171} C_VEL
LIN {X 0,Y 559.15,Z 238.459,A -85,B 0,C 180,E1 -3035.494,E2 -3035.494} C_VEL
LIN {X 0,Y 559.164,Z 238.453,A -85,B 0,C 180,E1 -3038.623,E2 -3038.623} C_VEL
LIN {X 0,Y 559.164,Z 238.453,A -85,B 0,C 180,E1 -3040.925,E2 -3040.925} C_VEL
LIN {X 0,Y 559.165,Z 238.457,A -85,B 0,C 180,E1 -3043.947,E2 -3043.947} C_VEL
LIN {X 0,Y 559.167,Z 238.454,A -85,B 0,C 180,E1 -3046.183,E2 -3046.183} C_VEL
LIN {X 0,Y 559.202,Z 238.45,A -85,B 0,C 180,E1 -3049.133,E2 -3049.133} C_VEL
LIN {X 0,Y 559.201,Z 238.448,A -85,B 0,C 180,E1 -3052.053,E2 -3052.053} C_VEL
LIN {X 0,Y 559.252,Z 238.445,A -85,B 0,C 180,E1 -3054.952,E2 -3054.952} C_VEL
LIN {X 0,Y 559.24,Z 238.446,A -85,B 0,C 180,E1 -3057.838,E2 -3057.838} C_VEL
LIN {X 0,Y 559.268,Z 238.442,A -85,B 0,C 180,E1 -3060.719,E2 -3060.719} C_VEL
LIN {X 0,Y 559.236,Z 238.448,A -85,B 0,C 180,E1 -3062.88,E2 -3062.88} C_VEL
LIN {X 0,Y 559.219,Z 238.447,A -85,B 0,C 180,E1 -3065.769,E2 -3065.769} C_VEL
LIN {X 0,Y 559.182,Z 238.454,A -85,B 0,C 180,E1 -3068.673,E2 -3068.673} C_VEL
LIN {X 0,Y 559.197,Z 238.451,A -85,B 0,C 180,E1 -3071.599,E2 -3071.599} C_VEL
LIN {X 0,Y 559.186,Z 238.453,A -85,B 0,C 180,E1 -3074.595,E2 -3074.595} C_VEL
LIN {X 0,Y 559.147,Z 238.456,A -85,B 0,C 180,E1 -3077.556,E2 -3077.556} C_VEL
LIN {X 0,Y 559.162,Z 238.453,A -85,B 0,C 180,E1 -3079.836,E2 -3079.836} C_VEL
LIN {X 0,Y 559.142,Z 238.457,A -85,B 0,C 180,E1 -3082.151,E2 -3082.151} C_VEL
LIN {X 0,Y 559.147,Z 238.46,A -85,B 0,C 180,E1 -3084.504,E2 -3084.504} C_VEL
LIN {X 0,Y 559.156,Z 238.46,A -85,B 0,C 180,E1 -3086.902,E2 -3086.902} C_VEL
LIN {X 0,Y 559.174,Z 238.451,A -85,B 0,C 180,E1 -3089.864,E2 -3089.864} C_VEL
LIN {X 0,Y 559.133,Z 238.457,A -85,B 0,C 180,E1 -3090.633,E2 -3090.633} C_VEL
LIN {X 0,Y 558.468,Z 238.541,A -85,B 0,C 180,E1 -3091.234,E2 -3091.234} C_VEL
LIN {X 0,Y 555.605,Z 238.899,A -85,B 0,C 180,E1 -3092.21,E2 -3092.21} C_VEL
LIN {X 0,Y 553.193,Z 239.2,A -85,B 0,C 180,E1 -3092.996,E2 -3092.996} C_VEL
LIN {X 0,Y 552.173,Z 239.324,A -85,B 0,C 180,E1 -3093.603,E2 -3093.603} C_VEL
LIN {X 0,Y 552.099,Z 239.334,A -85,B 0,C 180,E1 -3093.808,E2 -3093.808} C_VEL
LIN {X 0,Y 552.096,Z 239.34,A -85,B 0,C 180,E1 -3096.746,E2 -3096.746} C_VEL
LIN {X 0,Y 552.12,Z 239.33,A -85,B 0,C 180,E1 -3099.526,E2 -3099.526} C_VEL
LIN {X 0,Y 552.116,Z 239.339,A -85,B 0,C 180,E1 -3102.425,E2 -3102.425} C_VEL
LIN {X 0,Y 552.083,Z 239.336,A -85,B 0,C 180,E1 -3105.563,E2 -3105.563} C_VEL
LIN {X 0,Y 552.124,Z 239.335,A -85,B 0,C 180,E1 -3108.676,E2 -3108.676} C_VEL
LIN {X 0,Y 552.105,Z 239.336,A -85,B 0,C 180,E1 -3111.411,E2 -3111.411} C_VEL
LIN {X 0,Y 552.154,Z 239.385,A -85,B 0,C 180,E1 -3114.134,E2 -3114.134} C_VEL
LIN {X 0,Y 553.037,Z 245.153,A -85,B 0,C 180,E1 -3115.121,E2 -3115.121} C_VEL
LIN {X 0,Y 552.641,Z 262.456,A -85,B 0,C 180,E1 -3117.92,E2 -3117.92} C_VEL
LIN {X 0,Y 552.609,Z 267.043,A -85,B 0,C 180,E1 -3118.642,E2 -3118.642} C_VEL
LIN {X 0,Y 554.193,Z 275.942,A -85,B 0,C 180,E1 -3118.813,E2 -3118.813} C_VEL
LIN {X 0,Y 553.752,Z 403.869,A -85,B 0,C 180,E1 -3120.516,E2 -3120.516} C_VEL
LIN {X 0,Y 553.568,Z 417.708,A -85,B 0,C 180,E1 -3120.844,E2 -3120.844} C_VEL
LIN {X 0,Y 553.394,Z 430.554,A -85,B 0,C 180,E1 -3121.284,E2 -3121.284} C_VEL
LIN {X 0,Y 553.157,Z 443.287,A -85,B 0,C 180,E1 -3121.857,E2 -3121.857} C_VEL
LIN {X 0,Y 552.881,Z 455.63,A -85,B 0,C 180,E1 -3122.562,E2 -3122.562} C_VEL
LIN {X 0,Y 552.679,Z 467.105,A -85,B 0,C 180,E1 -3123.372,E2 -3123.372} C_VEL
LIN {X 0,Y 552.452,Z 478.737,A -85,B 0,C 180,E1 -3124.372,E2 -3124.372} C_VEL
LIN {X 0,Y 552.203,Z 488.325,A -85,B 0,C 180,E1 -3125.367,E2 -3125.367} C_VEL
LIN {X 0,Y 552.048,Z 498.063,A -85,B 0,C 180,E1 -3126.588,E2 -3126.588} C_VEL
LIN {X 0,Y 551.929,Z 505.617,A -85,B 0,C 180,E1 -3127.74,E2 -3127.74} C_VEL
LIN {X 0,Y 551.816,Z 512.925,A -85,B 0,C 180,E1 -3129.108,E2 -3129.108} C_VEL
LIN {X 0,Y 551.803,Z 518.625,A -85,B 0,C 180,E1 -3130.47,E2 -3130.47} C_VEL
LIN {X 0,Y 551.695,Z 522.889,A -85,B 0,C 180,E1 -3131.814,E2 -3131.814} C_VEL
LIN {X 0,Y 551.683,Z 525.517,A -85,B 0,C 180,E1 -3132.963,E2 -3132.963} C_VEL
LIN {X 0,Y 551.621,Z 527.725,A -85,B 0,C 180,E1 -3134.482,E2 -3134.482} C_VEL
LIN {X 0,Y 551.675,Z 528.495,A -85,B 0,C 180,E1 -3135.993,E2 -3135.993} C_VEL
LIN {X 0,Y 551.651,Z 527.848,A -85,B 0,C 180,E1 -3137.492,E2 -3137.492} C_VEL
LIN {X 0,Y 551.695,Z 525.796,A -85,B 0,C 180,E1 -3138.984,E2 -3138.984} C_VEL
LIN {X 0,Y 551.696,Z 522.33,A -85,B 0,C 180,E1 -3140.468,E2 -3140.468} C_VEL
LIN {X 0,Y 551.792,Z 517.362,A -85,B 0,C 180,E1 -3141.946,E2 -3141.946} C_VEL
LIN {X 0,Y 551.872,Z 510.771,A -85,B 0,C 180,E1 -3143.419,E2 -3143.419} C_VEL
LIN {X 0,Y 551.907,Z 503.481,A -85,B 0,C 180,E1 -3144.703,E2 -3144.703} C_VEL
LIN {X 0,Y 552.06,Z 495.864,A -85,B 0,C 180,E1 -3145.802,E2 -3145.802} C_VEL
LIN {X 0,Y 552.242,Z 486.769,A -85,B 0,C 180,E1 -3146.9,E2 -3146.9} C_VEL
LIN {X 0,Y 552.472,Z 475.785,A -85,B 0,C 180,E1 -3147.995,E2 -3147.995} C_VEL
LIN {X 0,Y 552.714,Z 464.647,A -85,B 0,C 180,E1 -3148.907,E2 -3148.907} C_VEL
LIN {X 0,Y 553.001,Z 452.383,A -85,B 0,C 180,E1 -3149.727,E2 -3149.727} C_VEL
LIN {X 0,Y 553.215,Z 440.644,A -85,B 0,C 180,E1 -3150.364,E2 -3150.364} C_VEL
LIN {X 0,Y 553.443,Z 426.607,A -85,B 0,C 180,E1 -3150.955,E2 -3150.955} C_VEL
LIN {X 0,Y 553.622,Z 412.458,A -85,B 0,C 180,E1 -3151.387,E2 -3151.387} C_VEL
LIN {X 0,Y 553.755,Z 398.684,A -85,B 0,C 180,E1 -3151.659,E2 -3151.659} C_VEL
LIN {X 0,Y 554.118,Z 274.782,A -85,B 0,C 180,E1 -3153.295,E2 -3153.295} C_VEL
LIN {X 0,Y 552.606,Z 266.836,A -85,B 0,C 180,E1 -3153.463,E2 -3153.463} C_VEL
LIN {X 0,Y 552.907,Z 249.829,A -85,B 0,C 180,E1 -3156.202,E2 -3156.202} C_VEL
LIN {X 0,Y 552.908,Z 243.114,A -85,B 0,C 180,E1 -3157.303,E2 -3157.303} C_VEL
LIN {X 0,Y 552.158,Z 239.336,A -85,B 0,C 180,E1 -3157.998,E2 -3157.998} C_VEL
LIN {X 0,Y 552.167,Z 239.326,A -85,B 0,C 180,E1 -3161.006,E2 -3161.006} C_VEL
LIN {X 0,Y 552.128,Z 239.34,A -85,B 0,C 180,E1 -3163.995,E2 -3163.995} C_VEL
LIN {X 0,Y 552.145,Z 239.327,A -85,B 0,C 180,E1 -3167.023,E2 -3167.023} C_VEL
LIN {X 0,Y 552.121,Z 239.334,A -85,B 0,C 180,E1 -3170.101,E2 -3170.101} C_VEL
LIN {X 0,Y 552.084,Z 239.335,A -85,B 0,C 180,E1 -3172.451,E2 -3172.451} C_VEL
LIN {X 0,Y 552.149,Z 239.336,A -85,B 0,C 180,E1 -3175.643,E2 -3175.643} C_VEL
LIN {X 0,Y 552.114,Z 239.331,A -85,B 0,C 180,E1 -3178.563,E2 -3178.563} C_VEL
LIN {X 0,Y 552.121,Z 239.338,A -85,B 0,C 180,E1 -3181.48,E2 -3181.48} C_VEL
LIN {X 0,Y 552.132,Z 239.33,A -85,B 0,C 180,E1 -3184.173,E2 -3184.173} C_VEL
LIN {X 0,Y 552.098,Z 239.334,A -85,B 0,C 180,E1 -3186.747,E2 -3186.747} C_VEL
LIN {X 0,Y 552.137,Z 239.336,A -85,B 0,C 180,E1 -3189.526,E2 -3189.526} C_VEL
LIN {X 0,Y 552.118,Z 239.33,A -85,B 0,C 180,E1 -3192.426,E2 -3192.426} C_VEL
LIN {X 0,Y 552.085,Z 239.34,A -85,B 0,C 180,E1 -3195.563,E2 -3195.563} C_VEL
LIN {X 0,Y 552.157,Z 239.327,A -85,B 0,C 180,E1 -3198.673,E2 -3198.673} C_VEL
LIN {X 0,Y 552.108,Z 239.338,A -85,B 0,C 180,E1 -3201.412,E2 -3201.412} C_VEL
LIN {X 0,Y 552.101,Z 239.332,A -85,B 0,C 180,E1 -3204.159,E2 -3204.159} C_VEL
LIN {X 0,Y 552.116,Z 239.336,A -85,B 0,C 180,E1 -3206.816,E2 -3206.816} C_VEL
LIN {X 0,Y 552.102,Z 239.337,A -85,B 0,C 180,E1 -3209.392,E2 -3209.392} C_VEL
LIN {X 0,Y 552.115,Z 239.331,A -85,B 0,C 180,E1 -3211.904,E2 -3211.904} C_VEL
LIN {X 0,Y 552.144,Z 239.332,A -85,B 0,C 180,E1 -3214.65,E2 -3214.65} C_VEL
LIN {X 0,Y 552.085,Z 239.336,A -85,B 0,C 180,E1 -3217.55,E2 -3217.55} C_VEL
LIN {X 0,Y 552.138,Z 239.331,A -85,B 0,C 180,E1 -3220.374,E2 -3220.374} C_VEL
LIN {X 0,Y 552.147,Z 239.333,A -85,B 0,C 180,E1 -3222.978,E2 -3222.978} C_VEL
LIN {X 0,Y 552.128,Z 239.33,A -85,B 0,C 180,E1 -3226.005,E2 -3226.005} C_VEL
LIN {X 0,Y 552.152,Z 239.331,A -85,B 0,C 180,E1 -3228.994,E2 -3228.994} C_VEL
LIN {X 0,Y 552.151,Z 239.327,A -85,B 0,C 180,E1 -3231.953,E2 -3231.953} C_VEL
LIN {X 0,Y 552.224,Z 239.322,A -85,B 0,C 180,E1 -3234.89,E2 -3234.89} C_VEL
LIN {X 0,Y 552.215,Z 239.319,A -85,B 0,C 180,E1 -3237.813,E2 -3237.813} C_VEL
LIN {X 0,Y 552.238,Z 239.321,A -85,B 0,C 180,E1 -3240.73,E2 -3240.73} C_VEL
LIN {X 0,Y 552.201,Z 239.323,A -85,B 0,C 180,E1 -3242.919,E2 -3242.919} C_VEL
LIN {X 0,Y 552.194,Z 239.323,A -85,B 0,C 180,E1 -3245.845,E2 -3245.845} C_VEL
LIN {X 0,Y 552.156,Z 239.328,A -85,B 0,C 180,E1 -3248.787,E2 -3248.787} C_VEL
LIN {X 0,Y 552.156,Z 239.328,A -85,B 0,C 180,E1 -3251.751,E2 -3251.751} C_VEL
LIN {X 0,Y 552.13,Z 239.331,A -85,B 0,C 180,E1 -3254.749,E2 -3254.749} C_VEL
LIN {X 0,Y 552.109,Z 239.335,A -85,B 0,C 180,E1 -3257.789,E2 -3257.789} C_VEL
LIN {X 0,Y 552.125,Z 239.339,A -85,B 0,C 180,E1 -3260.102,E2 -3260.102} C_VEL
LIN {X 0,Y 552.091,Z 239.338,A -85,B 0,C 180,E1 -3262.452,E2 -3262.452} C_VEL
LIN {X 0,Y 552.15,Z 239.327,A -85,B 0,C 180,E1 -3265.351,E2 -3265.351} C_VEL
LIN {X 0,Y 552.121,Z 239.338,A -85,B 0,C 180,E1 -3268.098,E2 -3268.098} C_VEL
LIN {X 0,Y 552.11,Z 239.332,A -85,B 0,C 180,E1 -3270.61,E2 -3270.61} C_VEL
LIN {X 0,Y 552.119,Z 239.331,A -85,B 0,C 180,E1 -3273.186,E2 -3273.186} C_VEL
LIN {X 0,Y 552.11,Z 239.341,A -85,B 0,C 180,E1 -3275.842,E2 -3275.842} C_VEL
LIN {X 0,Y 552.123,Z 239.33,A -85,B 0,C 180,E1 -3279.063,E2 -3279.063} C_VEL
LIN {X 0,Y 552.126,Z 239.334,A -85,B 0,C 180,E1 -3281.446,E2 -3281.446} C_VEL
LIN {X 0,Y 552.093,Z 239.334,A -85,B 0,C 180,E1 -3284.533,E2 -3284.533} C_VEL
LIN {X 0,Y 552.13,Z 239.338,A -85,B 0,C 180,E1 -3287.585,E2 -3287.585} C_VEL
LIN {X 0,Y 552.128,Z 239.329,A -85,B 0,C 180,E1 -3290.474,E2 -3290.474} C_VEL
LIN {X 0,Y 552.105,Z 239.338,A -85,B 0,C 180,E1 -3293.318,E2 -3293.318} C_VEL
LIN {X 0,Y 552.127,Z 239.332,A -85,B 0,C 180,E1 -3295.94,E2 -3295.94} C_VEL
LIN {X 0,Y 552.12,Z 239.333,A -85,B 0,C 180,E1 -3298.541,E2 -3298.541} C_VEL
LIN {X 0,Y 552.125,Z 239.339,A -85,B 0,C 180,E1 -3301.439,E2 -3301.439} C_VEL
LIN {X 0,Y 552.132,Z 239.334,A -85,B 0,C 180,E1 -3304.356,E2 -3304.356} C_VEL
LIN {X 0,Y 552.165,Z 239.436,A -85,B 0,C 180,E1 -3304.877,E2 -3304.877} C_VEL
LIN {X 0,Y 553.58,Z 247.203,A -85,B 0,C 180,E1 -3306.031,E2 -3306.031} C_VEL
LIN {X 0,Y 553.245,Z 267.192,A -85,B 0,C 180,E1 -3308.775,E2 -3308.775} C_VEL
LIN {X 0,Y 552.849,Z 290.022,A -85,B 0,C 180,E1 -3311.854,E2 -3311.854} C_VEL
LIN {X 0,Y 552.761,Z 295.551,A -85,B 0,C 180,E1 -3312.587,E2 -3312.587} C_VEL
LIN {X 0,Y 554.227,Z 303.913,A -85,B 0,C 180,E1 -3312.745,E2 -3312.745} C_VEL
LIN {X 0,Y 553.758,Z 433.897,A -85,B 0,C 180,E1 -3314.472,E2 -3314.472} C_VEL
LIN {X 0,Y 553.568,Z 448.518,A -85,B 0,C 180,E1 -3314.824,E2 -3314.824} C_VEL
LIN {X 0,Y 553.359,Z 462.839,A -85,B 0,C 180,E1 -3315.332,E2 -3315.332} C_VEL
LIN {X 0,Y 553.144,Z 475.641,A -85,B 0,C 180,E1 -3315.937,E2 -3315.937} C_VEL
LIN {X 0,Y 552.879,Z 488.101,A -85,B 0,C 180,E1 -3316.68,E2 -3316.68} C_VEL
LIN {X 0,Y 552.623,Z 500.651,A -85,B 0,C 180,E1 -3317.608,E2 -3317.608} C_VEL
LIN {X 0,Y 552.448,Z 511.296,A -85,B 0,C 180,E1 -3318.573,E2 -3318.573} C_VEL
LIN {X 0,Y 552.18,Z 521.853,A -85,B 0,C 180,E1 -3319.736,E2 -3319.736} C_VEL
LIN {X 0,Y 552.033,Z 530.175,A -85,B 0,C 180,E1 -3320.843,E2 -3320.843} C_VEL
LIN {X 0,Y 551.913,Z 538.127,A -85,B 0,C 180,E1 -3322.132,E2 -3322.132} C_VEL
LIN {X 0,Y 551.823,Z 544.528,A -85,B 0,C 180,E1 -3323.418,E2 -3323.418} C_VEL
LIN {X 0,Y 551.792,Z 548.961,A -85,B 0,C 180,E1 -3324.518,E2 -3324.518} C_VEL
LIN {X 0,Y 551.76,Z 552.444,A -85,B 0,C 180,E1 -3325.617,E2 -3325.617} C_VEL
LIN {X 0,Y 551.72,Z 555.832,A -85,B 0,C 180,E1 -3327.079,E2 -3327.079} C_VEL
LIN {X 0,Y 551.64,Z 557.834,A -85,B 0,C 180,E1 -3328.54,E2 -3328.54} C_VEL
LIN {X 0,Y 551.639,Z 558.5,A -85,B 0,C 180,E1 -3330,E2 -3330} C_VEL
LIN {X 0,Y 551.64,Z 557.836,A -85,B 0,C 180,E1 -3331.46,E2 -3331.46} C_VEL
LIN {X 0,Y 551.72,Z 555.836,A -85,B 0,C 180,E1 -3332.921,E2 -3332.921} C_VEL
LIN {X 0,Y 551.76,Z 552.447,A -85,B 0,C 180,E1 -3334.383,E2 -3334.383} C_VEL
LIN {X 0,Y 551.824,Z 547.568,A -85,B 0,C 180,E1 -3335.848,E2 -3335.848} C_VEL
LIN {X 0,Y 551.833,Z 541.055,A -85,B 0,C 180,E1 -3337.317,E2 -3337.317} C_VEL
LIN {X 0,Y 551.963,Z 533.805,A -85,B 0,C 180,E1 -3338.604,E2 -3338.604} C_VEL
LIN {X 0,Y 552.116,Z 524.824,A -85,B 0,C 180,E1 -3339.895,E2 -3339.895} C_VEL
LIN {X 0,Y 552.347,Z 515.396,A -85,B 0,C 180,E1 -3341.003,E2 -3341.003} C_VEL
LIN {X 0,Y 552.524,Z 504.956,A -85,B 0,C 180,E1 -3342.022,E2 -3342.022} C_VEL
LIN {X 0,Y 552.734,Z 493.433,A -85,B 0,C 180,E1 -3342.95,E2 -3342.95} C_VEL
LIN {X 0,Y 553.05,Z 480.645,A -85,B 0,C 180,E1 -3343.784,E2 -3343.784} C_VEL
LIN {X 0,Y 553.251,Z 468.153,A -85,B 0,C 180,E1 -3344.436,E2 -3344.436} C_VEL
LIN {X 0,Y 553.508,Z 455.085,A -85,B 0,C 180,E1 -3344.963,E2 -3344.963} C_VEL
LIN {X 0,Y 553.665,Z 441.464,A -85,B 0,C 180,E1 -3345.365,E2 -3345.365} C_VEL
LIN {X 0,Y 553.774,Z 426.632,A -85,B 0,C 180,E1 -3345.645,E2 -3345.645} C_VEL
LIN {X 0,Y 554.155,Z 303.268,A -85,B 0,C 180,E1 -3347.266,E2 -3347.266} C_VEL
LIN {X 0,Y 552.751,Z 295.389,A -85,B 0,C 180,E1 -3347.428,E2 -3347.428} C_VEL
LIN {X 0,Y 553.096,Z 274.302,A -85,B 0,C 180,E1 -3350.258,E2 -3350.258} C_VEL
LIN {X 0,Y 553.498,Z 252.858,A -85,B 0,C 180,E1 -3353.179,E2 -3353.179} C_VEL
LIN {X 0,Y 553.463,Z 245.733,A -85,B 0,C 180,E1 -3354.174,E2 -3354.174} C_VEL
LIN {X 0,Y 552.143,Z 239.335,A -85,B 0,C 180,E1 -3355.144,E2 -3355.144} C_VEL
LIN {X 0,Y 552.11,Z 239.336,A -85,B 0,C 180,E1 -3358.098,E2 -3358.098} C_VEL
LIN {X 0,Y 552.104,Z 239.342,A -85,B 0,C 180,E1 -3360.608,E2 -3360.608} C_VEL
LIN {X 0,Y 552.122,Z 239.334,A -85,B 0,C 180,E1 -3363.184,E2 -3363.184} C_VEL
LIN {X 0,Y 552.084,Z 239.339,A -85,B 0,C 180,E1 -3365.843,E2 -3365.843} C_VEL
LIN {X 0,Y 552.115,Z 239.339,A -85,B 0,C 180,E1 -3368.588,E2 -3368.588} C_VEL
LIN {X 0,Y 552.13,Z 239.329,A -85,B 0,C 180,E1 -3371.444,E2 -3371.444} C_VEL
LIN {X 0,Y 552.094,Z 239.339,A -85,B 0,C 180,E1 -3374.531,E2 -3374.531} C_VEL
LIN {X 0,Y 552.128,Z 239.331,A -85,B 0,C 180,E1 -3377.583,E2 -3377.583} C_VEL
LIN {X 0,Y 552.131,Z 239.334,A -85,B 0,C 180,E1 -3380.472,E2 -3380.472} C_VEL
LIN {X 0,Y 552.111,Z 239.331,A -85,B 0,C 180,E1 -3383.315,E2 -3383.315} C_VEL
LIN {X 0,Y 552.127,Z 239.335,A -85,B 0,C 180,E1 -3385.938,E2 -3385.938} C_VEL
LIN {X 0,Y 552.113,Z 239.331,A -85,B 0,C 180,E1 -3388.54,E2 -3388.54} C_VEL
LIN {X 0,Y 552.12,Z 239.333,A -85,B 0,C 180,E1 -3391.436,E2 -3391.436} C_VEL
LIN {X 0,Y 552.124,Z 239.332,A -85,B 0,C 180,E1 -3394.355,E2 -3394.355} C_VEL
LIN {X 0,Y 552.103,Z 239.332,A -85,B 0,C 180,E1 -3396.757,E2 -3396.757} C_VEL
LIN {X 0,Y 552.114,Z 239.333,A -85,B 0,C 180,E1 -3399.119,E2 -3399.119} C_VEL
LIN {X 0,Y 552.124,Z 239.335,A -85,B 0,C 180,E1 -3401.444,E2 -3401.444} C_VEL
LIN {X 0,Y 552.115,Z 239.338,A -85,B 0,C 180,E1 -3403.736,E2 -3403.736} C_VEL
LIN {X 0,Y 552.13,Z 239.333,A -85,B 0,C 180,E1 -3406.003,E2 -3406.003} C_VEL
LIN {X 0,Y 552.169,Z 239.325,A -85,B 0,C 180,E1 -3408.993,E2 -3408.993} C_VEL
LIN {X 0,Y 552.155,Z 239.327,A -85,B 0,C 180,E1 -3411.951,E2 -3411.951} C_VEL
LIN {X 0,Y 552.226,Z 239.32,A -85,B 0,C 180,E1 -3414.888,E2 -3414.888} C_VEL
LIN {X 0,Y 552.212,Z 239.321,A -85,B 0,C 180,E1 -3417.811,E2 -3417.811} C_VEL
LIN {X 0,Y 552.238,Z 239.317,A -85,B 0,C 180,E1 -3420.728,E2 -3420.728} C_VEL
LIN {X 0,Y 552.202,Z 239.324,A -85,B 0,C 180,E1 -3422.917,E2 -3422.917} C_VEL
LIN {X 0,Y 552.188,Z 239.322,A -85,B 0,C 180,E1 -3425.843,E2 -3425.843} C_VEL
LIN {X 0,Y 552.152,Z 239.331,A -85,B 0,C 180,E1 -3428.785,E2 -3428.785} C_VEL
LIN {X 0,Y 552.153,Z 239.327,A -85,B 0,C 180,E1 -3431.75,E2 -3431.75} C_VEL
LIN {X 0,Y 552.124,Z 239.335,A -85,B 0,C 180,E1 -3434.748,E2 -3434.748} C_VEL
LIN {X 0,Y 552.098,Z 239.333,A -85,B 0,C 180,E1 -3437.788,E2 -3437.788} C_VEL
LIN {X 0,Y 552.121,Z 239.331,A -85,B 0,C 180,E1 -3440.1,E2 -3440.1} C_VEL
LIN {X 0,Y 552.101,Z 239.337,A -85,B 0,C 180,E1 -3442.449,E2 -3442.449} C_VEL
LIN {X 0,Y 552.141,Z 239.33,A -85,B 0,C 180,E1 -3445.35,E2 -3445.35} C_VEL
LIN {X 0,Y 552.112,Z 239.333,A -85,B 0,C 180,E1 -3448.097,E2 -3448.097} C_VEL
LIN {X 0,Y 552.094,Z 239.338,A -85,B 0,C 180,E1 -3450.628,E2 -3450.628} C_VEL
LIN {X 0,Y 552.107,Z 239.334,A -85,B 0,C 180,E1 -3453.185,E2 -3453.185} C_VEL
LIN {X 0,Y 552.099,Z 239.334,A -85,B 0,C 180,E1 -3453.808,E2 -3453.808} C_VEL
LIN {X 0,Y 551.463,Z 239.42,A -85,B 0,C 180,E1 -3454.417,E2 -3454.417} C_VEL
LIN {X 0,Y 548.64,Z 239.773,A -85,B 0,C 180,E1 -3455.405,E2 -3455.405} C_VEL
LIN {X 0,Y 546.219,Z 240.074,A -85,B 0,C 180,E1 -3456.2,E2 -3456.2} C_VEL
LIN {X 0,Y 545.15,Z 240.205,A -85,B 0,C 180,E1 -3456.814,E2 -3456.814} C_VEL
LIN {X 0,Y 545.048,Z 240.214,A -85,B 0,C 180,E1 -3457.022,E2 -3457.022} C_VEL
LIN {X 0,Y 545.078,Z 240.212,A -85,B 0,C 180,E1 -3460.14,E2 -3460.14} C_VEL
LIN {X 0,Y 545.073,Z 240.21,A -85,B 0,C 180,E1 -3463.105,E2 -3463.105} C_VEL
LIN {X 0,Y 545.048,Z 240.221,A -85,B 0,C 180,E1 -3466.224,E2 -3466.224} C_VEL
LIN {X 0,Y 545.086,Z 240.21,A -85,B 0,C 180,E1 -3468.887,E2 -3468.887} C_VEL
LIN {X 0,Y 545.039,Z 240.22,A -85,B 0,C 180,E1 -3471.763,E2 -3471.763} C_VEL
LIN {X 0,Y 545.085,Z 240.296,A -85,B 0,C 180,E1 -3473.961,E2 -3473.961} C_VEL
LIN {X 0,Y 546.102,Z 246.656,A -85,B 0,C 180,E1 -3475.064,E2 -3475.064} C_VEL
LIN {X 0,Y 545.713,Z 262.72,A -85,B 0,C 180,E1 -3477.694,E2 -3477.694} C_VEL
LIN {X 0,Y 545.63,Z 267.156,A -85,B 0,C 180,E1 -3478.411,E2 -3478.411} C_VEL
LIN {X 0,Y 547.42,Z 276.617,A -85,B 0,C 180,E1 -3478.599,E2 -3478.599} C_VEL
LIN {X 0,Y 546.929,Z 402.937,A -85,B 0,C 180,E1 -3480.296,E2 -3480.296} C_VEL
LIN {X 0,Y 546.743,Z 417.228,A -85,B 0,C 180,E1 -3480.629,E2 -3480.629} C_VEL
LIN {X 0,Y 546.535,Z 431.078,A -85,B 0,C 180,E1 -3481.109,E2 -3481.109} C_VEL
LIN {X 0,Y 546.259,Z 443.53,A -85,B 0,C 180,E1 -3481.679,E2 -3481.679} C_VEL
LIN {X 0,Y 545.972,Z 455.828,A -85,B 0,C 180,E1 -3482.394,E2 -3482.394} C_VEL
LIN {X 0,Y 545.693,Z 468.479,A -85,B 0,C 180,E1 -3483.311,E2 -3483.311} C_VEL
LIN {X 0,Y 545.462,Z 479.262,A -85,B 0,C 180,E1 -3484.268,E2 -3484.268} C_VEL
LIN {X 0,Y 545.16,Z 490.112,A -85,B 0,C 180,E1 -3485.434,E2 -3485.434} C_VEL
LIN {X 0,Y 544.99,Z 499.311,A -85,B 0,C 180,E1 -3486.639,E2 -3486.639} C_VEL
LIN {X 0,Y 544.837,Z 506.821,A -85,B 0,C 180,E1 -3487.834,E2 -3487.834} C_VEL
LIN {X 0,Y 544.712,Z 513.841,A -85,B 0,C 180,E1 -3489.219,E2 -3489.219} C_VEL
LIN {X 0,Y 544.717,Z 518.638,A -85,B 0,C 180,E1 -3490.4,E2 -3490.4} C_VEL
LIN {X 0,Y 544.611,Z 522.347,A -85,B 0,C 180,E1 -3491.569,E2 -3491.569} C_VEL
LIN {X 0,Y 544.596,Z 525.147,A -85,B 0,C 180,E1 -3492.734,E2 -3492.734} C_VEL
LIN {X 0,Y 544.543,Z 527.524,A -85,B 0,C 180,E1 -3494.275,E2 -3494.275} C_VEL
LIN {X 0,Y 544.602,Z 528.456,A -85,B 0,C 180,E1 -3495.807,E2 -3495.807} C_VEL
LIN {X 0,Y 544.56,Z 527.985,A -85,B 0,C 180,E1 -3497.327,E2 -3497.327} C_VEL
LIN {X 0,Y 544.597,Z 526.13,A -85,B 0,C 180,E1 -3498.839,E2 -3498.839} C_VEL
LIN {X 0,Y 544.611,Z 522.853,A -85,B 0,C 180,E1 -3500.343,E2 -3500.343} C_VEL
LIN {X 0,Y 544.688,Z 518.063,A -85,B 0,C 180,E1 -3501.841,E2 -3501.841} C_VEL
LIN {X 0,Y 544.784,Z 511.657,A -85,B 0,C 180,E1 -3503.333,E2 -3503.333} C_VEL
LIN {X 0,Y 544.815,Z 504.573,A -85,B 0,C 180,E1 -3504.634,E2 -3504.634} C_VEL
LIN {X 0,Y 545.008,Z 497.177,A -85,B 0,C 180,E1 -3505.748,E2 -3505.748} C_VEL
LIN {X 0,Y 545.187,Z 488.347,A -85,B 0,C 180,E1 -3506.86,E2 -3506.86} C_VEL
LIN {X 0,Y 545.445,Z 477.744,A -85,B 0,C 180,E1 -3507.97,E2 -3507.97} C_VEL
LIN {X 0,Y 545.742,Z 465.906,A -85,B 0,C 180,E1 -3508.986,E2 -3508.986} C_VEL
LIN {X 0,Y 546.075,Z 453.967,A -85,B 0,C 180,E1 -3509.816,E2 -3509.816} C_VEL
LIN {X 0,Y 546.344,Z 440.692,A -85,B 0,C 180,E1 -3510.553,E2 -3510.553} C_VEL
LIN {X 0,Y 546.573,Z 427.905,A -85,B 0,C 180,E1 -3511.105,E2 -3511.105} C_VEL
LIN {X 0,Y 546.779,Z 414.194,A -85,B 0,C 180,E1 -3511.542,E2 -3511.542} C_VEL
LIN {X 0,Y 546.927,Z 399.955,A -85,B 0,C 180,E1 -3511.841,E2 -3511.841} C_VEL
LIN {X 0,Y 547.394,Z 276.212,A -85,B 0,C 180,E1 -3513.496,E2 -3513.496} C_VEL
LIN {X 0,Y 545.671,Z 267.03,A -85,B 0,C 180,E1 -3513.692,E2 -3513.692} C_VEL
LIN {X 0,Y 545.968,Z 251.126,A -85,B 0,C 180,E1 -3516.282,E2 -3516.282} C_VEL
LIN {X 0,Y 545.943,Z 244.419,A -85,B 0,C 180,E1 -3517.396,E2 -3517.396} C_VEL
LIN {X 0,Y 545.124,Z 240.212,A -85,B 0,C 180,E1 -3518.153,E2 -3518.153} C_VEL
LIN {X 0,Y 545.12,Z 240.205,A -85,B 0,C 180,E1 -3521.15,E2 -3521.15} C_VEL
LIN {X 0,Y 545.085,Z 240.214,A -85,B 0,C 180,E1 -3524.18,E2 -3524.18} C_VEL
LIN {X 0,Y 545.08,Z 240.211,A -85,B 0,C 180,E1 -3527.429,E2 -3527.429} C_VEL
LIN {X 0,Y 545.086,Z 240.208,A -85,B 0,C 180,E1 -3530.372,E2 -3530.372} C_VEL
LIN {X 0,Y 545.078,Z 240.214,A -85,B 0,C 180,E1 -3533.559,E2 -3533.559} C_VEL
LIN {X 0,Y 545.088,Z 240.21,A -85,B 0,C 180,E1 -3536,E2 -3536} C_VEL
LIN {X 0,Y 545.08,Z 240.207,A -85,B 0,C 180,E1 -3538.75,E2 -3538.75} C_VEL
LIN {X 0,Y 545.064,Z 240.217,A -85,B 0,C 180,E1 -3541.683,E2 -3541.683} C_VEL
LIN {X 0,Y 545.071,Z 240.208,A -85,B 0,C 180,E1 -3544.563,E2 -3544.563} C_VEL
LIN {X 0,Y 545.026,Z 240.221,A -85,B 0,C 180,E1 -3547.304,E2 -3547.304} C_VEL
LIN {X 0,Y 545.081,Z 240.208,A -85,B 0,C 180,E1 -3550.14,E2 -3550.14} C_VEL
LIN {X 0,Y 545.054,Z 240.211,A -85,B 0,C 180,E1 -3552.698,E2 -3552.698} C_VEL
LIN {X 0,Y 545.049,Z 240.218,A -85,B 0,C 180,E1 -3555.167,E2 -3555.167} C_VEL
LIN {X 0,Y 545.078,Z 240.209,A -85,B 0,C 180,E1 -3557.899,E2 -3557.899} C_VEL
LIN {X 0,Y 545.072,Z 240.212,A -85,B 0,C 180,E1 -3560.819,E2 -3560.819} C_VEL
LIN {X 0,Y 545.047,Z 240.214,A -85,B 0,C 180,E1 -3563.622,E2 -3563.622} C_VEL
LIN {X 0,Y 545.065,Z 240.209,A -85,B 0,C 180,E1 -3566.33,E2 -3566.33} C_VEL
LIN {X 0,Y 545.058,Z 240.218,A -85,B 0,C 180,E1 -3568.953,E2 -3568.953} C_VEL
LIN {X 0,Y 545.093,Z 240.208,A -85,B 0,C 180,E1 -3571.509,E2 -3571.509} C_VEL
LIN {X 0,Y 545.087,Z 240.209,A -85,B 0,C 180,E1 -3574.491,E2 -3574.491} C_VEL
LIN {X 0,Y 545.033,Z 240.217,A -85,B 0,C 180,E1 -3577.243,E2 -3577.243} C_VEL
LIN {X 0,Y 545.109,Z 240.207,A -85,B 0,C 180,E1 -3580.416,E2 -3580.416} C_VEL
LIN {X 0,Y 545.067,Z 240.209,A -85,B 0,C 180,E1 -3583.522,E2 -3583.522} C_VEL
LIN {X 0,Y 545.086,Z 240.206,A -85,B 0,C 180,E1 -3585.821,E2 -3585.821} C_VEL
LIN {X 0,Y 545.108,Z 240.211,A -85,B 0,C 180,E1 -3588.85,E2 -3588.85} C_VEL
LIN {X 0,Y 545.122,Z 240.202,A -85,B 0,C 180,E1 -3591.848,E2 -3591.848} C_VEL
LIN {X 0,Y 545.199,Z 240.198,A -85,B 0,C 180,E1 -3594.824,E2 -3594.824} C_VEL
LIN {X 0,Y 545.187,Z 240.194,A -85,B 0,C 180,E1 -3597.785,E2 -3597.785} C_VEL
LIN {X 0,Y 545.207,Z 240.197,A -85,B 0,C 180,E1 -3600.74,E2 -3600.74} C_VEL
LIN {X 0,Y 545.168,Z 240.198,A -85,B 0,C 180,E1 -3602.957,E2 -3602.957} C_VEL
LIN {X 0,Y 545.165,Z 240.199,A -85,B 0,C 180,E1 -3605.92,E2 -3605.92} C_VEL
LIN {X 0,Y 545.115,Z 240.204,A -85,B 0,C 180,E1 -3608.901,E2 -3608.901} C_VEL
LIN {X 0,Y 545.128,Z 240.205,A -85,B 0,C 180,E1 -3611.905,E2 -3611.905} C_VEL
LIN {X 0,Y 545.079,Z 240.208,A -85,B 0,C 180,E1 -3614.945,E2 -3614.945} C_VEL
LIN {X 0,Y 545.077,Z 240.215,A -85,B 0,C 180,E1 -3618.027,E2 -3618.027} C_VEL
LIN {X 0,Y 545.09,Z 240.211,A -85,B 0,C 180,E1 -3620.373,E2 -3620.373} C_VEL
LIN {X 0,Y 545.086,Z 240.209,A -85,B 0,C 180,E1 -3623.56,E2 -3623.56} C_VEL
LIN {X 0,Y 545.075,Z 240.217,A -85,B 0,C 180,E1 -3626.001,E2 -3626.001} C_VEL
LIN {X 0,Y 545.087,Z 240.206,A -85,B 0,C 180,E1 -3628.75,E2 -3628.75} C_VEL
LIN {X 0,Y 545.075,Z 240.214,A -85,B 0,C 180,E1 -3631.683,E2 -3631.683} C_VEL
LIN {X 0,Y 545.078,Z 240.208,A -85,B 0,C 180,E1 -3634.564,E2 -3634.564} C_VEL
LIN {X 0,Y 545.037,Z 240.215,A -85,B 0,C 180,E1 -3637.305,E2 -3637.305} C_VEL
LIN {X 0,Y 545.069,Z 240.212,A -85,B 0,C 180,E1 -3640.143,E2 -3640.143} C_VEL
LIN {X 0,Y 545.076,Z 240.209,A -85,B 0,C 180,E1 -3643.107,E2 -3643.107} C_VEL
LIN {X 0,Y 545.066,Z 240.21,A -85,B 0,C 180,E1 -3646.225,E2 -3646.225} C_VEL
LIN {X 0,Y 545.086,Z 240.207,A -85,B 0,C 180,E1 -3648.887,E2 -3648.887} C_VEL
LIN {X 0,Y 545.051,Z 240.217,A -85,B 0,C 180,E1 -3651.763,E2 -3651.763} C_VEL
LIN {X 0,Y 545.036,Z 240.212,A -85,B 0,C 180,E1 -3654.532,E2 -3654.532} C_VEL
LIN {X 0,Y 545.082,Z 240.213,A -85,B 0,C 180,E1 -3657.213,E2 -3657.213} C_VEL
LIN {X 0,Y 545.064,Z 240.215,A -85,B 0,C 180,E1 -3659.811,E2 -3659.811} C_VEL
LIN {X 0,Y 545.082,Z 240.21,A -85,B 0,C 180,E1 -3662.344,E2 -3662.344} C_VEL
LIN {X 0,Y 545.139,Z 240.317,A -85,B 0,C 180,E1 -3664.679,E2 -3664.679} C_VEL
LIN {X 0,Y 546.692,Z 248.31,A -85,B 0,C 180,E1 -3665.888,E2 -3665.888} C_VEL
LIN {X 0,Y 546.301,Z 268.45,A -85,B 0,C 180,E1 -3668.69,E2 -3668.69} C_VEL
LIN {X 0,Y 545.863,Z 291.258,A -85,B 0,C 180,E1 -3671.807,E2 -3671.807} C_VEL
LIN {X 0,Y 545.783,Z 295.31,A -85,B 0,C 180,E1 -3672.357,E2 -3672.357} C_VEL
LIN {X 0,Y 547.455,Z 305.849,A -85,B 0,C 180,E1 -3672.554,E2 -3672.554} C_VEL
LIN {X 0,Y 546.918,Z 433.681,A -85,B 0,C 180,E1 -3674.273,E2 -3674.273} C_VEL
LIN {X 0,Y 546.728,Z 447.44,A -85,B 0,C 180,E1 -3674.602,E2 -3674.602} C_VEL
LIN {X 0,Y 546.522,Z 461.568,A -85,B 0,C 180,E1 -3675.097,E2 -3675.097} C_VEL
LIN {X 0,Y 546.253,Z 473.771,A -85,B 0,C 180,E1 -3675.661,E2 -3675.661} C_VEL
LIN {X 0,Y 545.975,Z 486.615,A -85,B 0,C 180,E1 -3676.413,E2 -3676.413} C_VEL
LIN {X 0,Y 545.667,Z 498.295,A -85,B 0,C 180,E1 -3677.258,E2 -3677.258} C_VEL
LIN {X 0,Y 545.451,Z 509.119,A -85,B 0,C 180,E1 -3678.213,E2 -3678.213} C_VEL
LIN {X 0,Y 545.232,Z 518.707,A -85,B 0,C 180,E1 -3679.228,E2 -3679.228} C_VEL
LIN {X 0,Y 545.024,Z 527.557,A -85,B 0,C 180,E1 -3680.35,E2 -3680.35} C_VEL
LIN {X 0,Y 544.873,Z 536.034,A -85,B 0,C 180,E1 -3681.657,E2 -3681.657} C_VEL
LIN {X 0,Y 544.737,Z 542.864,A -85,B 0,C 180,E1 -3682.96,E2 -3682.96} C_VEL
LIN {X 0,Y 544.732,Z 547.569,A -85,B 0,C 180,E1 -3684.076,E2 -3684.076} C_VEL
LIN {X 0,Y 544.654,Z 552.444,A -85,B 0,C 180,E1 -3685.56,E2 -3685.56} C_VEL
LIN {X 0,Y 544.647,Z 555.832,A -85,B 0,C 180,E1 -3687.041,E2 -3687.041} C_VEL
LIN {X 0,Y 544.542,Z 557.835,A -85,B 0,C 180,E1 -3688.521,E2 -3688.521} C_VEL
LIN {X 0,Y 544.54,Z 558.5,A -85,B 0,C 180,E1 -3690,E2 -3690} C_VEL
LIN {X 0,Y 544.542,Z 557.836,A -85,B 0,C 180,E1 -3691.479,E2 -3691.479} C_VEL
LIN {X 0,Y 544.647,Z 555.836,A -85,B 0,C 180,E1 -3692.958,E2 -3692.958} C_VEL
LIN {X 0,Y 544.654,Z 552.447,A -85,B 0,C 180,E1 -3694.44,E2 -3694.44} C_VEL
LIN {X 0,Y 544.736,Z 547.568,A -85,B 0,C 180,E1 -3695.924,E2 -3695.924} C_VEL
LIN {X 0,Y 544.784,Z 541.055,A -85,B 0,C 180,E1 -3697.412,E2 -3697.412} C_VEL
LIN {X 0,Y 544.911,Z 533.805,A -85,B 0,C 180,E1 -3698.716,E2 -3698.716} C_VEL
LIN {X 0,Y 545.082,Z 524.824,A -85,B 0,C 180,E1 -3700.024,E2 -3700.024} C_VEL
LIN {X 0,Y 545.35,Z 515.395,A -85,B 0,C 180,E1 -3701.145,E2 -3701.145} C_VEL
LIN {X 0,Y 545.546,Z 504.955,A -85,B 0,C 180,E1 -3702.178,E2 -3702.178} C_VEL
LIN {X 0,Y 545.794,Z 493.397,A -85,B 0,C 180,E1 -3703.117,E2 -3703.117} C_VEL
LIN {X 0,Y 546.117,Z 480.559,A -85,B 0,C 180,E1 -3703.963,E2 -3703.963} C_VEL
LIN {X 0,Y 546.378,Z 468.022,A -85,B 0,C 180,E1 -3704.621,E2 -3704.621} C_VEL
LIN {X 0,Y 546.674,Z 454.047,A -85,B 0,C 180,E1 -3705.186,E2 -3705.186} C_VEL
LIN {X 0,Y 546.846,Z 439.87,A -85,B 0,C 180,E1 -3705.598,E2 -3705.598} C_VEL
LIN {X 0,Y 546.967,Z 424.595,A -85,B 0,C 180,E1 -3705.869,E2 -3705.869} C_VEL
LIN {X 0,Y 547.373,Z 304.297,A -85,B 0,C 180,E1 -3707.469,E2 -3707.469} C_VEL
LIN {X 0,Y 545.8,Z 295.148,A -85,B 0,C 180,E1 -3707.661,E2 -3707.661} C_VEL
LIN {X 0,Y 546.155,Z 274.117,A -85,B 0,C 180,E1 -3710.527,E2 -3710.527} C_VEL
LIN {X 0,Y 546.623,Z 252.696,A -85,B 0,C 180,E1 -3713.488,E2 -3713.488} C_VEL
LIN {X 0,Y 546.506,Z 246.991,A -85,B 0,C 180,E1 -3714.299,E2 -3714.299} C_VEL
LIN {X 0,Y 545.12,Z 240.209,A -85,B 0,C 180,E1 -3715.343,E2 -3715.343} C_VEL
LIN {X 0,Y 545.102,Z 240.214,A -85,B 0,C 180,E1 -3718.492,E2 -3718.492} C_VEL
LIN {X 0,Y 545.067,Z 240.214,A -85,B 0,C 180,E1 -3721.047,E2 -3721.047} C_VEL
LIN {X 0,Y 545.068,Z 240.213,A -85,B 0,C 180,E1 -3723.671,E2 -3723.671} C_VEL
LIN {X 0,Y 545.068,Z 240.212,A -85,B 0,C 180,E1 -3726.925,E2 -3726.925} C_VEL
LIN {X 0,Y 545.064,Z 240.218,A -85,B 0,C 180,E1 -3730.142,E2 -3730.142} C_VEL
LIN {X 0,Y 545.084,Z 240.208,A -85,B 0,C 180,E1 -3733.105,E2 -3733.105} C_VEL
LIN {X 0,Y 545.053,Z 240.219,A -85,B 0,C 180,E1 -3736.224,E2 -3736.224} C_VEL
LIN {X 0,Y 545.094,Z 240.207,A -85,B 0,C 180,E1 -3738.886,E2 -3738.886} C_VEL
LIN {X 0,Y 545.05,Z 240.216,A -85,B 0,C 180,E1 -3741.762,E2 -3741.762} C_VEL
LIN {X 0,Y 545.06,Z 240.209,A -85,B 0,C 180,E1 -3744.533,E2 -3744.533} C_VEL
LIN {X 0,Y 545.076,Z 240.208,A -85,B 0,C 180,E1 -3747.211,E2 -3747.211} C_VEL
LIN {X 0,Y 545.097,Z 240.211,A -85,B 0,C 180,E1 -3749.812,E2 -3749.812} C_VEL
LIN {X 0,Y 545.091,Z 240.205,A -85,B 0,C 180,E1 -3752.825,E2 -3752.825} C_VEL
LIN {X 0,Y 545.046,Z 240.218,A -85,B 0,C 180,E1 -3755.63,E2 -3755.63} C_VEL
LIN {X 0,Y 545.059,Z 240.21,A -85,B 0,C 180,E1 -3758.836,E2 -3758.836} C_VEL
LIN {X 0,Y 545.077,Z 240.21,A -85,B 0,C 180,E1 -3761.195,E2 -3761.195} C_VEL
LIN {X 0,Y 545.071,Z 240.216,A -85,B 0,C 180,E1 -3763.52,E2 -3763.52} C_VEL
LIN {X 0,Y 545.088,Z 240.212,A -85,B 0,C 180,E1 -3765.819,E2 -3765.819} C_VEL
LIN {X 0,Y 545.124,Z 240.201,A -85,B 0,C 180,E1 -3768.849,E2 -3768.849} C_VEL
LIN {X 0,Y 545.126,Z 240.203,A -85,B 0,C 180,E1 -3771.846,E2 -3771.846} C_VEL
LIN {X 0,Y 545.201,Z 240.194,A -85,B 0,C 180,E1 -3774.822,E2 -3774.822} C_VEL
LIN {X 0,Y 545.184,Z 240.197,A -85,B 0,C 180,E1 -3777.783,E2 -3777.783} C_VEL
LIN {X 0,Y 545.207,Z 240.193,A -85,B 0,C 180,E1 -3780.738,E2 -3780.738} C_VEL
LIN {X 0,Y 545.168,Z 240.201,A -85,B 0,C 180,E1 -3782.955,E2 -3782.955} C_VEL
LIN {X 0,Y 545.16,Z 240.197,A -85,B 0,C 180,E1 -3785.919,E2 -3785.919} C_VEL
LIN {X 0,Y 545.111,Z 240.21,A -85,B 0,C 180,E1 -3788.899,E2 -3788.899} C_VEL
LIN {X 0,Y 545.124,Z 240.202,A -85,B 0,C 180,E1 -3791.903,E2 -3791.903} C_VEL
LIN {X 0,Y 545.073,Z 240.217,A -85,B 0,C 180,E1 -3794.943,E2 -3794.943} C_VEL
LIN {X 0,Y 545.067,Z 240.209,A -85,B 0,C 180,E1 -3798.025,E2 -3798.025} C_VEL
LIN {X 0,Y 545.086,Z 240.209,A -85,B 0,C 180,E1 -3800.371,E2 -3800.371} C_VEL
LIN {X 0,Y 545.101,Z 240.204,A -85,B 0,C 180,E1 -3803.557,E2 -3803.557} C_VEL
LIN {X 0,Y 545.065,Z 240.21,A -85,B 0,C 180,E1 -3806,E2 -3806} C_VEL
LIN {X 0,Y 545.079,Z 240.215,A -85,B 0,C 180,E1 -3808.749,E2 -3808.749} C_VEL
LIN {X 0,Y 545.054,Z 240.212,A -85,B 0,C 180,E1 -3811.047,E2 -3811.047} C_VEL
LIN {X 0,Y 545.05,Z 240.212,A -85,B 0,C 180,E1 -3813.807,E2 -3813.807} C_VEL
LIN {X 0,Y 545.059,Z 240.214,A -85,B 0,C 180,E1 -3816.926,E2 -3816.926} C_VEL
LIN {X 0,Y 545.048,Z 240.214,A -85,B 0,C 180,E1 -3817.022,E2 -3817.022} C_VEL
LIN {X 0,Y 544.343,Z 240.301,A -85,B 0,C 180,E1 -3817.639,E2 -3817.639} C_VEL
LIN {X 0,Y 541.49,Z 240.659,A -85,B 0,C 180,E1 -3818.64,E2 -3818.64} C_VEL
LIN {X 0,Y 539.112,Z 240.952,A -85,B 0,C 180,E1 -3819.446,E2 -3819.446} C_VEL
LIN {X 0,Y 538.108,Z 241.08,A -85,B 0,C 180,E1 -3820.068,E2 -3820.068} C_VEL
LIN {X 0,Y 538.033,Z 241.086,A -85,B 0,C 180,E1 -3820.278,E2 -3820.278} C_VEL
LIN {X 0,Y 538.019,Z 241.09,A -85,B 0,C 180,E1 -3822.988,E2 -3822.988} C_VEL
LIN {X 0,Y 538.013,Z 241.093,A -85,B 0,C 180,E1 -3825.925,E2 -3825.925} C_VEL
LIN {X 0,Y 538.063,Z 241.084,A -85,B 0,C 180,E1 -3829.249,E2 -3829.249} C_VEL
LIN {X 0,Y 537.979,Z 241.101,A -85,B 0,C 180,E1 -3832.122,E2 -3832.122} C_VEL
LIN {X 0,Y 538.069,Z 241.122,A -85,B 0,C 180,E1 -3833.771,E2 -3833.771} C_VEL
LIN {X 0,Y 539.192,Z 248.152,A -85,B 0,C 180,E1 -3835.006,E2 -3835.006} C_VEL
LIN {X 0,Y 538.771,Z 264.267,A -85,B 0,C 180,E1 -3837.669,E2 -3837.669} C_VEL
LIN {X 0,Y 538.747,Z 267.649,A -85,B 0,C 180,E1 -3838.182,E2 -3838.182} C_VEL
LIN {X 0,Y 540.615,Z 276.957,A -85,B 0,C 180,E1 -3838.375,E2 -3838.375} C_VEL
LIN {X 0,Y 540.098,Z 403.392,A -85,B 0,C 180,E1 -3840.097,E2 -3840.097} C_VEL
LIN {X 0,Y 539.898,Z 417.965,A -85,B 0,C 180,E1 -3840.447,E2 -3840.447} C_VEL
LIN {X 0,Y 539.69,Z 431.603,A -85,B 0,C 180,E1 -3840.93,E2 -3840.93} C_VEL
LIN {X 0,Y 539.372,Z 443.806,A -85,B 0,C 180,E1 -3841.497,E2 -3841.497} C_VEL
LIN {X 0,Y 539.034,Z 457.034,A -85,B 0,C 180,E1 -3842.283,E2 -3842.283} C_VEL
LIN {X 0,Y 538.758,Z 468.73,A -85,B 0,C 180,E1 -3843.149,E2 -3843.149} C_VEL
LIN {X 0,Y 538.467,Z 479.971,A -85,B 0,C 180,E1 -3844.164,E2 -3844.164} C_VEL
LIN {X 0,Y 538.158,Z 490.33,A -85,B 0,C 180,E1 -3845.299,E2 -3845.299} C_VEL
LIN {X 0,Y 537.972,Z 499.475,A -85,B 0,C 180,E1 -3846.519,E2 -3846.519} C_VEL
LIN {X 0,Y 537.79,Z 506.935,A -85,B 0,C 180,E1 -3847.73,E2 -3847.73} C_VEL
LIN {X 0,Y 537.686,Z 513.018,A -85,B 0,C 180,E1 -3848.934,E2 -3848.934} C_VEL
LIN {X 0,Y 537.632,Z 518.358,A -85,B 0,C 180,E1 -3850.248,E2 -3850.248} C_VEL
LIN {X 0,Y 537.505,Z 522.916,A -85,B 0,C 180,E1 -3851.712,E2 -3851.712} C_VEL
LIN {X 0,Y 537.516,Z 525.046,A -85,B 0,C 180,E1 -3852.638,E2 -3852.638} C_VEL
LIN {X 0,Y 537.443,Z 527.32,A -85,B 0,C 180,E1 -3854.062,E2 -3854.062} C_VEL
LIN {X 0,Y 537.505,Z 528.415,A -85,B 0,C 180,E1 -3855.616,E2 -3855.616} C_VEL
LIN {X 0,Y 537.465,Z 528.104,A -85,B 0,C 180,E1 -3857.157,E2 -3857.157} C_VEL
LIN {X 0,Y 537.521,Z 526.407,A -85,B 0,C 180,E1 -3858.69,E2 -3858.69} C_VEL
LIN {X 0,Y 537.503,Z 523.317,A -85,B 0,C 180,E1 -3860.214,E2 -3860.214} C_VEL
LIN {X 0,Y 537.606,Z 518.765,A -85,B 0,C 180,E1 -3861.732,E2 -3861.732} C_VEL
LIN {X 0,Y 537.634,Z 514.29,A -85,B 0,C 180,E1 -3862.867,E2 -3862.867} C_VEL
LIN {X 0,Y 537.787,Z 508.848,A -85,B 0,C 180,E1 -3863.999,E2 -3863.999} C_VEL
LIN {X 0,Y 537.924,Z 501.121,A -85,B 0,C 180,E1 -3865.316,E2 -3865.316} C_VEL
LIN {X 0,Y 538.074,Z 493.09,A -85,B 0,C 180,E1 -3866.443,E2 -3866.443} C_VEL
LIN {X 0,Y 538.386,Z 483.429,A -85,B 0,C 180,E1 -3867.569,E2 -3867.569} C_VEL
LIN {X 0,Y 538.619,Z 472.782,A -85,B 0,C 180,E1 -3868.598,E2 -3868.598} C_VEL
LIN {X 0,Y 538.977,Z 460.994,A -85,B 0,C 180,E1 -3869.533,E2 -3869.533} C_VEL
LIN {X 0,Y 539.271,Z 449.444,A -85,B 0,C 180,E1 -3870.28,E2 -3870.28} C_VEL
LIN {X 0,Y 539.569,Z 435.891,A -85,B 0,C 180,E1 -3870.98,E2 -3870.98} C_VEL
LIN {X 0,Y 539.835,Z 422.032,A -85,B 0,C 180,E1 -3871.515,E2 -3871.515} C_VEL
LIN {X 0,Y 540.012,Z 408.474,A -85,B 0,C 180,E1 -3871.888,E2 -3871.888} C_VEL
LIN {X 0,Y 540.167,Z 393.299,A -85,B 0,C 180,E1 -3872.144,E2 -3872.144} C_VEL
LIN {X 0,Y 540.631,Z 276.897,A -85,B 0,C 180,E1 -3873.715,E2 -3873.715} C_VEL
LIN {X 0,Y 538.73,Z 267.229,A -85,B 0,C 180,E1 -3873.927,E2 -3873.927} C_VEL
LIN {X 0,Y 539.048,Z 251.303,A -85,B 0,C 180,E1 -3876.551,E2 -3876.551} C_VEL
LIN {X 0,Y 539.111,Z 246.367,A -85,B 0,C 180,E1 -3877.377,E2 -3877.377} C_VEL
LIN {X 0,Y 538.091,Z 241.087,A -85,B 0,C 180,E1 -3878.331,E2 -3878.331} C_VEL
LIN {X 0,Y 538.084,Z 241.086,A -85,B 0,C 180,E1 -3881.605,E2 -3881.605} C_VEL
LIN {X 0,Y 538.044,Z 241.087,A -85,B 0,C 180,E1 -3884.858,E2 -3884.858} C_VEL
LIN {X 0,Y 538.044,Z 241.089,A -85,B 0,C 180,E1 -3887.541,E2 -3887.541} C_VEL
LIN {X 0,Y 538.029,Z 241.085,A -85,B 0,C 180,E1 -3890.651,E2 -3890.651} C_VEL
LIN {X 0,Y 538.027,Z 241.092,A -85,B 0,C 180,E1 -3893.887,E2 -3893.887} C_VEL
LIN {X 0,Y 538.043,Z 241.084,A -85,B 0,C 180,E1 -3896.366,E2 -3896.366} C_VEL
LIN {X 0,Y 538.042,Z 241.085,A -85,B 0,C 180,E1 -3898.939,E2 -3898.939} C_VEL
LIN {X 0,Y 538.014,Z 241.091,A -85,B 0,C 180,E1 -3901.891,E2 -3901.891} C_VEL
LIN {X 0,Y 538.021,Z 241.087,A -85,B 0,C 180,E1 -3904.622,E2 -3904.622} C_VEL
LIN {X 0,Y 537.994,Z 241.095,A -85,B 0,C 180,E1 -3907.171,E2 -3907.171} C_VEL
LIN {X 0,Y 538.044,Z 241.087,A -85,B 0,C 180,E1 -3909.794,E2 -3909.794} C_VEL
LIN {X 0,Y 538.011,Z 241.089,A -85,B 0,C 180,E1 -3912.786,E2 -3912.786} C_VEL
LIN {X 0,Y 538.016,Z 241.088,A -85,B 0,C 180,E1 -3915.926,E2 -3915.926} C_VEL
LIN {X 0,Y 538.067,Z 241.09,A -85,B 0,C 180,E1 -3919.249,E2 -3919.249} C_VEL
LIN {X 0,Y 537.982,Z 241.091,A -85,B 0,C 180,E1 -3922.123,E2 -3922.123} C_VEL
LIN {X 0,Y 538.009,Z 241.094,A -85,B 0,C 180,E1 -3924.918,E2 -3924.918} C_VEL
LIN {X 0,Y 538.019,Z 241.089,A -85,B 0,C 180,E1 -3927.619,E2 -3927.619} C_VEL
LIN {X 0,Y 538.03,Z 241.086,A -85,B 0,C 180,E1 -3930.241,E2 -3930.241} C_VEL
LIN {X 0,Y 538.06,Z 241.088,A -85,B 0,C 180,E1 -3932.797,E2 -3932.797} C_VEL
LIN {X 0,Y 538.037,Z 241.088,A -85,B 0,C 180,E1 -3935.294,E2 -3935.294} C_VEL
LIN {X 0,Y 538.003,Z 241.089,A -85,B 0,C 180,E1 -3938.043,E2 -3938.043} C_VEL
LIN {X 0,Y 538.03,Z 241.093,A -85,B 0,C 180,E1 -3940.941,E2 -3940.941} C_VEL
LIN {X 0,Y 538.017,Z 241.089,A -85,B 0,C 180,E1 -3943.3,E2 -3943.3} C_VEL
LIN {X 0,Y 538.054,Z 241.082,A -85,B 0,C 180,E1 -3945.632,E2 -3945.632} C_VEL
LIN {X 0,Y 538.067,Z 241.09,A -85,B 0,C 180,E1 -3948.703,E2 -3948.703} C_VEL
LIN {X 0,Y 538.078,Z 241.079,A -85,B 0,C 180,E1 -3951.741,E2 -3951.741} C_VEL
LIN {X 0,Y 538.175,Z 241.074,A -85,B 0,C 180,E1 -3954.756,E2 -3954.756} C_VEL
LIN {X 0,Y 538.159,Z 241.07,A -85,B 0,C 180,E1 -3957.756,E2 -3957.756} C_VEL
LIN {X 0,Y 538.177,Z 241.072,A -85,B 0,C 180,E1 -3960.749,E2 -3960.749} C_VEL
LIN {X 0,Y 538.134,Z 241.074,A -85,B 0,C 180,E1 -3962.995,E2 -3962.995} C_VEL
LIN {X 0,Y 538.118,Z 241.078,A -85,B 0,C 180,E1 -3965.998,E2 -3965.998} C_VEL
LIN {X 0,Y 538.065,Z 241.082,A -85,B 0,C 180,E1 -3969.019,E2 -3969.019} C_VEL
LIN {X 0,Y 538.077,Z 241.086,A -85,B 0,C 180,E1 -3972.064,E2 -3972.064} C_VEL
LIN {X 0,Y 538.039,Z 241.084,A -85,B 0,C 180,E1 -3975.145,E2 -3975.145} C_VEL
LIN {X 0,Y 538.029,Z 241.093,A -85,B 0,C 180,E1 -3978.271,E2 -3978.271} C_VEL
LIN {X 0,Y 538.034,Z 241.087,A -85,B 0,C 180,E1 -3980.652,E2 -3980.652} C_VEL
LIN {X 0,Y 538.019,Z 241.093,A -85,B 0,C 180,E1 -3983.888,E2 -3983.888} C_VEL
LIN {X 0,Y 538.038,Z 241.088,A -85,B 0,C 180,E1 -3986.368,E2 -3986.368} C_VEL
LIN {X 0,Y 538.033,Z 241.085,A -85,B 0,C 180,E1 -3988.936,E2 -3988.936} C_VEL
LIN {X 0,Y 538.024,Z 241.095,A -85,B 0,C 180,E1 -3991.891,E2 -3991.891} C_VEL
LIN {X 0,Y 538.028,Z 241.086,A -85,B 0,C 180,E1 -3994.622,E2 -3994.622} C_VEL
LIN {X 0,Y 538.005,Z 241.09,A -85,B 0,C 180,E1 -3997.171,E2 -3997.171} C_VEL
LIN {X 0,Y 538.026,Z 241.095,A -85,B 0,C 180,E1 -3999.797,E2 -3999.797} C_VEL
LIN {X 0,Y 538.016,Z 241.087,A -85,B 0,C 180,E1 -4002.787,E2 -4002.787} C_VEL
LIN {X 0,Y 538.029,Z 241.09,A -85,B 0,C 180,E1 -4005.926,E2 -4005.926} C_VEL
LIN {X 0,Y 538.048,Z 241.087,A -85,B 0,C 180,E1 -4009.254,E2 -4009.254} C_VEL
LIN {X 0,Y 537.991,Z 241.092,A -85,B 0,C 180,E1 -4012.123,E2 -4012.123} C_VEL
LIN {X 0,Y 537.998,Z 241.091,A -85,B 0,C 180,E1 -4014.916,E2 -4014.916} C_VEL
LIN {X 0,Y 538.027,Z 241.096,A -85,B 0,C 180,E1 -4017.619,E2 -4017.619} C_VEL
LIN {X 0,Y 538.018,Z 241.09,A -85,B 0,C 180,E1 -4020.24,E2 -4020.24} C_VEL
LIN {X 0,Y 538.058,Z 241.087,A -85,B 0,C 180,E1 -4022.796,E2 -4022.796} C_VEL
LIN {X 0,Y 538.073,Z 241.162,A -85,B 0,C 180,E1 -4024.468,E2 -4024.468} C_VEL
LIN {X 0,Y 539.811,Z 250.137,A -85,B 0,C 180,E1 -4025.844,E2 -4025.844} C_VEL
LIN {X 0,Y 539.37,Z 269.695,A -85,B 0,C 180,E1 -4028.603,E2 -4028.603} C_VEL
LIN {X 0,Y 538.885,Z 292.482,A -85,B 0,C 180,E1 -4031.76,E2 -4031.76} C_VEL
LIN {X 0,Y 538.868,Z 295.053,A -85,B 0,C 180,E1 -4032.114,E2 -4032.114} C_VEL
LIN {X 0,Y 540.674,Z 306.252,A -85,B 0,C 180,E1 -4032.336,E2 -4032.336} C_VEL
LIN {X 0,Y 540.086,Z 433.439,A -85,B 0,C 180,E1 -4034.069,E2 -4034.069} C_VEL
LIN {X 0,Y 539.868,Z 448.018,A -85,B 0,C 180,E1 -4034.427,E2 -4034.427} C_VEL
LIN {X 0,Y 539.605,Z 462.48,A -85,B 0,C 180,E1 -4034.95,E2 -4034.95} C_VEL
LIN {X 0,Y 539.315,Z 475.326,A -85,B 0,C 180,E1 -4035.569,E2 -4035.569} C_VEL
LIN {X 0,Y 538.981,Z 487.834,A -85,B 0,C 180,E1 -4036.33,E2 -4036.33} C_VEL
LIN {X 0,Y 538.676,Z 500.443,A -85,B 0,C 180,E1 -4037.282,E2 -4037.282} C_VEL
LIN {X 0,Y 538.387,Z 510.921,A -85,B 0,C 180,E1 -4038.248,E2 -4038.248} C_VEL
LIN {X 0,Y 538.139,Z 521.752,A -85,B 0,C 180,E1 -4039.465,E2 -4039.465} C_VEL
LIN {X 0,Y 537.943,Z 530.122,A -85,B 0,C 180,E1 -4040.601,E2 -4040.601} C_VEL
LIN {X 0,Y 537.757,Z 538.122,A -85,B 0,C 180,E1 -4041.924,E2 -4041.924} C_VEL
LIN {X 0,Y 537.668,Z 544.528,A -85,B 0,C 180,E1 -4043.244,E2 -4043.244} C_VEL
LIN {X 0,Y 537.579,Z 550.201,A -85,B 0,C 180,E1 -4044.749,E2 -4044.749} C_VEL
LIN {X 0,Y 537.576,Z 554.316,A -85,B 0,C 180,E1 -4046.252,E2 -4046.252} C_VEL
LIN {X 0,Y 537.489,Z 557.003,A -85,B 0,C 180,E1 -4047.752,E2 -4047.752} C_VEL
LIN {X 0,Y 537.439,Z 558.334,A -85,B 0,C 180,E1 -4049.251,E2 -4049.251} C_VEL
LIN {X 0,Y 537.439,Z 558.334,A -85,B 0,C 180,E1 -4050.749,E2 -4050.749} C_VEL
LIN {X 0,Y 537.489,Z 557.006,A -85,B 0,C 180,E1 -4052.248,E2 -4052.248} C_VEL
LIN {X 0,Y 537.576,Z 554.32,A -85,B 0,C 180,E1 -4053.748,E2 -4053.748} C_VEL
LIN {X 0,Y 537.579,Z 550.202,A -85,B 0,C 180,E1 -4055.251,E2 -4055.251} C_VEL
LIN {X 0,Y 537.673,Z 545.274,A -85,B 0,C 180,E1 -4056.581,E2 -4056.581} C_VEL
LIN {X 0,Y 537.764,Z 539.134,A -85,B 0,C 180,E1 -4057.887,E2 -4057.887} C_VEL
LIN {X 0,Y 537.911,Z 531.36,A -85,B 0,C 180,E1 -4059.21,E2 -4059.21} C_VEL
LIN {X 0,Y 538.096,Z 523.243,A -85,B 0,C 180,E1 -4060.345,E2 -4060.345} C_VEL
LIN {X 0,Y 538.352,Z 513.937,A -85,B 0,C 180,E1 -4061.433,E2 -4061.433} C_VEL
LIN {X 0,Y 538.612,Z 502.609,A -85,B 0,C 180,E1 -4062.528,E2 -4062.528} C_VEL
LIN {X 0,Y 538.93,Z 490.585,A -85,B 0,C 180,E1 -4063.479,E2 -4063.479} C_VEL
LIN {X 0,Y 539.257,Z 478.748,A -85,B 0,C 180,E1 -4064.24,E2 -4064.24} C_VEL
LIN {X 0,Y 539.496,Z 465.797,A -85,B 0,C 180,E1 -4064.908,E2 -4064.908} C_VEL
LIN {X 0,Y 539.801,Z 451.609,A -85,B 0,C 180,E1 -4065.46,E2 -4065.46} C_VEL
LIN {X 0,Y 540.055,Z 437.616,A -85,B 0,C 180,E1 -4065.843,E2 -4065.843} C_VEL
LIN {X 0,Y 540.148,Z 422.525,A -85,B 0,C 180,E1 -4066.099,E2 -4066.099} C_VEL
LIN {X 0,Y 540.662,Z 306.079,A -85,B 0,C 180,E1 -4067.666,E2 -4067.666} C_VEL
LIN {X 0,Y 538.861,Z 294.967,A -85,B 0,C 180,E1 -4067.892,E2 -4067.892} C_VEL
LIN {X 0,Y 539.308,Z 271.055,A -85,B 0,C 180,E1 -4071.199,E2 -4071.199} C_VEL
LIN {X 0,Y 539.759,Z 252.52,A -85,B 0,C 180,E1 -4073.805,E2 -4073.805} C_VEL
LIN {X 0,Y 539.597,Z 248.453,A -85,B 0,C 180,E1 -4074.395,E2 -4074.395} C_VEL
LIN {X 0,Y 538.072,Z 241.087,A -85,B 0,C 180,E1 -4075.532,E2 -4075.532} C_VEL
LIN {X 0,Y 538.04,Z 241.088,A -85,B 0,C 180,E1 -4078.049,E2 -4078.049} C_VEL
LIN {X 0,Y 538.021,Z 241.096,A -85,B 0,C 180,E1 -4080.626,E2 -4080.626} C_VEL
LIN {X 0,Y 538.045,Z 241.088,A -85,B 0,C 180,E1 -4083.282,E2 -4083.282} C_VEL
LIN {X 0,Y 537.993,Z 241.096,A -85,B 0,C 180,E1 -4086.004,E2 -4086.004} C_VEL
LIN {X 0,Y 538.011,Z 241.094,A -85,B 0,C 180,E1 -4088.83,E2 -4088.83} C_VEL
LIN {X 0,Y 538.035,Z 241.086,A -85,B 0,C 180,E1 -4091.772,E2 -4091.772} C_VEL
LIN {X 0,Y 538.029,Z 241.088,A -85,B 0,C 180,E1 -4094.858,E2 -4094.858} C_VEL
LIN {X 0,Y 538.035,Z 241.093,A -85,B 0,C 180,E1 -4098.119,E2 -4098.119} C_VEL
LIN {X 0,Y 538.036,Z 241.09,A -85,B 0,C 180,E1 -4100.413,E2 -4100.413} C_VEL
LIN {X 0,Y 538.025,Z 241.084,A -85,B 0,C 180,E1 -4103.066,E2 -4103.066} C_VEL
LIN {X 0,Y 538.023,Z 241.089,A -85,B 0,C 180,E1 -4105.826,E2 -4105.826} C_VEL
LIN {X 0,Y 538.019,Z 241.087,A -85,B 0,C 180,E1 -4108.499,E2 -4108.499} C_VEL
LIN {X 0,Y 538.054,Z 241.083,A -85,B 0,C 180,E1 -4111.099,E2 -4111.099} C_VEL
LIN {X 0,Y 538.037,Z 241.09,A -85,B 0,C 180,E1 -4113.632,E2 -4113.632} C_VEL
LIN {X 0,Y 538.016,Z 241.091,A -85,B 0,C 180,E1 -4116.117,E2 -4116.117} C_VEL
LIN {X 0,Y 538.032,Z 241.089,A -85,B 0,C 180,E1 -4119.348,E2 -4119.348} C_VEL
LIN {X 0,Y 538.065,Z 241.081,A -85,B 0,C 180,E1 -4122.517,E2 -4122.517} C_VEL
LIN {X 0,Y 538.056,Z 241.092,A -85,B 0,C 180,E1 -4125.63,E2 -4125.63} C_VEL
LIN {X 0,Y 538.081,Z 241.078,A -85,B 0,C 180,E1 -4128.701,E2 -4128.701} C_VEL
LIN {X 0,Y 538.082,Z 241.082,A -85,B 0,C 180,E1 -4131.739,E2 -4131.739} C_VEL
LIN {X 0,Y 538.158,Z 241.071,A -85,B 0,C 180,E1 -4134.754,E2 -4134.754} C_VEL
LIN {X 0,Y 538.156,Z 241.073,A -85,B 0,C 180,E1 -4137.754,E2 -4137.754} C_VEL
LIN {X 0,Y 538.177,Z 241.069,A -85,B 0,C 180,E1 -4140.747,E2 -4140.747} C_VEL
LIN {X 0,Y 538.134,Z 241.078,A -85,B 0,C 180,E1 -4142.993,E2 -4142.993} C_VEL
LIN {X 0,Y 538.113,Z 241.074,A -85,B 0,C 180,E1 -4145.996,E2 -4145.996} C_VEL
LIN {X 0,Y 538.062,Z 241.09,A -85,B 0,C 180,E1 -4149.017,E2 -4149.017} C_VEL
LIN {X 0,Y 538.072,Z 241.081,A -85,B 0,C 180,E1 -4152.062,E2 -4152.062} C_VEL
LIN {X 0,Y 538.033,Z 241.092,A -85,B 0,C 180,E1 -4155.143,E2 -4155.143} C_VEL
LIN {X 0,Y 538.019,Z 241.088,A -85,B 0,C 180,E1 -4158.269,E2 -4158.269} C_VEL
LIN {X 0,Y 538.03,Z 241.092,A -85,B 0,C 180,E1 -4160.65,E2 -4160.65} C_VEL
LIN {X 0,Y 538.028,Z 241.085,A -85,B 0,C 180,E1 -4163.886,E2 -4163.886} C_VEL
LIN {X 0,Y 538.028,Z 241.091,A -85,B 0,C 180,E1 -4166.366,E2 -4166.366} C_VEL
LIN {X 0,Y 538.042,Z 241.088,A -85,B 0,C 180,E1 -4168.938,E2 -4168.938} C_VEL
LIN {X 0,Y 537.999,Z 241.089,A -85,B 0,C 180,E1 -4171.887,E2 -4171.887} C_VEL
LIN {X 0,Y 538.012,Z 241.092,A -85,B 0,C 180,E1 -4174.62,E2 -4174.62} C_VEL
LIN {X 0,Y 537.992,Z 241.092,A -85,B 0,C 180,E1 -4177.17,E2 -4177.17} C_VEL
LIN {X 0,Y 538.033,Z 241.086,A -85,B 0,C 180,E1 -4180.278,E2 -4180.278} C_VEL
LIN {X 0,Y 537.382,Z 241.171,A -85,B 0,C 180,E1 -4180.903,E2 -4180.903} C_VEL
LIN {X 0,Y 534.522,Z 241.526,A -85,B 0,C 180,E1 -4181.918,E2 -4181.918} C_VEL
LIN {X 0,Y 532.089,Z 241.831,A -85,B 0,C 180,E1 -4182.735,E2 -4182.735} C_VEL
LIN {X 0,Y 531.037,Z 241.959,A -85,B 0,C 180,E1 -4183.366,E2 -4183.366} C_VEL
LIN {X 0,Y 530.949,Z 241.969,A -85,B 0,C 180,E1 -4183.579,E2 -4183.579} C_VEL
LIN {X 0,Y 530.95,Z 241.975,A -85,B 0,C 180,E1 -4186.505,E2 -4186.505} C_VEL
LIN {X 0,Y 530.993,Z 241.966,A -85,B 0,C 180,E1 -4189.569,E2 -4189.569} C_VEL
LIN {X 0,Y 530.953,Z 241.976,A -85,B 0,C 180,E1 -4192.576,E2 -4192.576} C_VEL
LIN {X 0,Y 531.021,Z 242.021,A -85,B 0,C 180,E1 -4193.585,E2 -4193.585} C_VEL
LIN {X 0,Y 532.259,Z 249.679,A -85,B 0,C 180,E1 -4194.947,E2 -4194.947} C_VEL
LIN {X 0,Y 531.833,Z 265.082,A -85,B 0,C 180,E1 -4197.521,E2 -4197.521} C_VEL
LIN {X 0,Y 531.812,Z 267.738,A -85,B 0,C 180,E1 -4197.94,E2 -4197.94} C_VEL
LIN {X 0,Y 533.885,Z 277.984,A -85,B 0,C 180,E1 -4198.156,E2 -4198.156} C_VEL
LIN {X 0,Y 533.296,Z 403.868,A -85,B 0,C 180,E1 -4199.895,E2 -4199.895} C_VEL
LIN {X 0,Y 533.057,Z 418.541,A -85,B 0,C 180,E1 -4200.255,E2 -4200.255} C_VEL
LIN {X 0,Y 532.838,Z 432.106,A -85,B 0,C 180,E1 -4200.745,E2 -4200.745} C_VEL
LIN {X 0,Y 532.49,Z 444.081,A -85,B 0,C 180,E1 -4201.31,E2 -4201.31} C_VEL
LIN {X 0,Y 532.173,Z 456.831,A -85,B 0,C 180,E1 -4202.076,E2 -4202.076} C_VEL
LIN {X 0,Y 531.814,Z 468.977,A -85,B 0,C 180,E1 -4202.983,E2 -4202.983} C_VEL
LIN {X 0,Y 531.512,Z 479.505,A -85,B 0,C 180,E1 -4203.94,E2 -4203.94} C_VEL
LIN {X 0,Y 531.215,Z 488.825,A -85,B 0,C 180,E1 -4204.954,E2 -4204.954} C_VEL
LIN {X 0,Y 530.976,Z 498.55,A -85,B 0,C 180,E1 -4206.231,E2 -4206.231} C_VEL
LIN {X 0,Y 530.759,Z 505.984,A -85,B 0,C 180,E1 -4207.419,E2 -4207.419} C_VEL
LIN {X 0,Y 530.637,Z 512.285,A -85,B 0,C 180,E1 -4208.641,E2 -4208.641} C_VEL
LIN {X 0,Y 530.547,Z 518.421,A -85,B 0,C 180,E1 -4210.133,E2 -4210.133} C_VEL
LIN {X 0,Y 530.466,Z 522.561,A -85,B 0,C 180,E1 -4211.46,E2 -4211.46} C_VEL
LIN {X 0,Y 530.385,Z 526.082,A -85,B 0,C 180,E1 -4213.052,E2 -4213.052} C_VEL
LIN {X 0,Y 530.357,Z 528.07,A -85,B 0,C 180,E1 -4214.632,E2 -4214.632} C_VEL
LIN {X 0,Y 530.396,Z 528.613,A -85,B 0,C 180,E1 -4216.202,E2 -4216.202} C_VEL
LIN {X 0,Y 530.368,Z 527.775,A -85,B 0,C 180,E1 -4217.76,E2 -4217.76} C_VEL
LIN {X 0,Y 530.411,Z 525.56,A -85,B 0,C 180,E1 -4219.31,E2 -4219.31} C_VEL
LIN {X 0,Y 530.442,Z 521.94,A -85,B 0,C 180,E1 -4220.852,E2 -4220.852} C_VEL
LIN {X 0,Y 530.562,Z 516.819,A -85,B 0,C 180,E1 -4222.388,E2 -4222.388} C_VEL
LIN {X 0,Y 530.664,Z 511.62,A -85,B 0,C 180,E1 -4223.589,E2 -4223.589} C_VEL
LIN {X 0,Y 530.754,Z 504.813,A -85,B 0,C 180,E1 -4224.872,E2 -4224.872} C_VEL
LIN {X 0,Y 530.958,Z 497.449,A -85,B 0,C 180,E1 -4226.015,E2 -4226.015} C_VEL
LIN {X 0,Y 531.203,Z 488.644,A -85,B 0,C 180,E1 -4227.156,E2 -4227.156} C_VEL
LIN {X 0,Y 531.506,Z 478.032,A -85,B 0,C 180,E1 -4228.295,E2 -4228.295} C_VEL
LIN {X 0,Y 531.845,Z 467.314,A -85,B 0,C 180,E1 -4229.243,E2 -4229.243} C_VEL
LIN {X 0,Y 532.251,Z 455.602,A -85,B 0,C 180,E1 -4230.095,E2 -4230.095} C_VEL
LIN {X 0,Y 532.58,Z 442.74,A -85,B 0,C 180,E1 -4230.851,E2 -4230.851} C_VEL
LIN {X 0,Y 532.894,Z 429.215,A -85,B 0,C 180,E1 -4231.464,E2 -4231.464} C_VEL
LIN {X 0,Y 533.121,Z 415.009,A -85,B 0,C 180,E1 -4231.936,E2 -4231.936} C_VEL
LIN {X 0,Y 533.296,Z 401.04,A -85,B 0,C 180,E1 -4232.242,E2 -4232.242} C_VEL
LIN {X 0,Y 533.899,Z 279.233,A -85,B 0,C 180,E1 -4233.916,E2 -4233.916} C_VEL
LIN {X 0,Y 532.685,Z 271.837,A -85,B 0,C 180,E1 -4234.061,E2 -4234.061} C_VEL
LIN {X 0,Y 531.79,Z 267.429,A -85,B 0,C 180,E1 -4234.168,E2 -4234.168} C_VEL
LIN {X 0,Y 532.124,Z 252.646,A -85,B 0,C 180,E1 -4236.636,E2 -4236.636} C_VEL
LIN {X 0,Y 532.144,Z 247.674,A -85,B 0,C 180,E1 -4237.474,E2 -4237.474} C_VEL
LIN {X 0,Y 531.057,Z 241.962,A -85,B 0,C 180,E1 -4238.514,E2 -4238.514} C_VEL
LIN {X 0,Y 531.045,Z 241.964,A -85,B 0,C 180,E1 -4241.677,E2 -4241.677} C_VEL
LIN {X 0,Y 531.016,Z 241.963,A -85,B 0,C 180,E1 -4244.956,E2 -4244.956} C_VEL
LIN {X 0,Y 531.002,Z 241.969,A -85,B 0,C 180,E1 -4247.723,E2 -4247.723} C_VEL
LIN {X 0,Y 530.988,Z 241.963,A -85,B 0,C 180,E1 -4250.938,E2 -4250.938} C_VEL
LIN {X 0,Y 530.975,Z 241.966,A -85,B 0,C 180,E1 -4254.224,E2 -4254.224} C_VEL
LIN {X 0,Y 531.001,Z 241.961,A -85,B 0,C 180,E1 -4256.743,E2 -4256.743} C_VEL
LIN {X 0,Y 530.986,Z 241.968,A -85,B 0,C 180,E1 -4259.322,E2 -4259.322} C_VEL
LIN {X 0,Y 530.967,Z 241.967,A -85,B 0,C 180,E1 -4262.104,E2 -4262.104} C_VEL
LIN {X 0,Y 530.977,Z 241.965,A -85,B 0,C 180,E1 -4264.855,E2 -4264.855} C_VEL
LIN {X 0,Y 530.952,Z 241.976,A -85,B 0,C 180,E1 -4267.508,E2 -4267.508} C_VEL
LIN {X 0,Y 531.014,Z 241.959,A -85,B 0,C 180,E1 -4270.429,E2 -4270.429} C_VEL
LIN {X 0,Y 530.954,Z 241.974,A -85,B 0,C 180,E1 -4273.495,E2 -4273.495} C_VEL
LIN {X 0,Y 530.954,Z 241.967,A -85,B 0,C 180,E1 -4276.506,E2 -4276.506} C_VEL
LIN {X 0,Y 530.996,Z 241.966,A -85,B 0,C 180,E1 -4279.57,E2 -4279.57} C_VEL
LIN {X 0,Y 530.957,Z 241.968,A -85,B 0,C 180,E1 -4282.577,E2 -4282.577} C_VEL
LIN {X 0,Y 530.992,Z 241.968,A -85,B 0,C 180,E1 -4285.312,E2 -4285.312} C_VEL
LIN {X 0,Y 530.969,Z 241.965,A -85,B 0,C 180,E1 -4288.034,E2 -4288.034} C_VEL
LIN {X 0,Y 530.994,Z 241.969,A -85,B 0,C 180,E1 -4290.871,E2 -4290.871} C_VEL
LIN {X 0,Y 531,Z 241.966,A -85,B 0,C 180,E1 -4293.258,E2 -4293.258} C_VEL
LIN {X 0,Y 530.985,Z 241.963,A -85,B 0,C 180,E1 -4295.958,E2 -4295.958} C_VEL
LIN {X 0,Y 530.991,Z 241.969,A -85,B 0,C 180,E1 -4299.063,E2 -4299.063} C_VEL
LIN {X 0,Y 531.005,Z 241.962,A -85,B 0,C 180,E1 -4302.279,E2 -4302.279} C_VEL
LIN {X 0,Y 531.008,Z 241.961,A -85,B 0,C 180,E1 -4305.437,E2 -4305.437} C_VEL
LIN {X 0,Y 531.026,Z 241.965,A -85,B 0,C 180,E1 -4308.551,E2 -4308.551} C_VEL
LIN {X 0,Y 531.048,Z 241.955,A -85,B 0,C 180,E1 -4311.63,E2 -4311.63} C_VEL
LIN {X 0,Y 531.131,Z 241.953,A -85,B 0,C 180,E1 -4314.686,E2 -4314.686} C_VEL
LIN {X 0,Y 531.131,Z 241.945,A -85,B 0,C 180,E1 -4317.726,E2 -4317.726} C_VEL
LIN {X 0,Y 531.147,Z 241.948,A -85,B 0,C 180,E1 -4320.759,E2 -4320.759} C_VEL
LIN {X 0,Y 531.1,Z 241.95,A -85,B 0,C 180,E1 -4323.035,E2 -4323.035} C_VEL
LIN {X 0,Y 531.077,Z 241.956,A -85,B 0,C 180,E1 -4326.078,E2 -4326.078} C_VEL
LIN {X 0,Y 531.025,Z 241.958,A -85,B 0,C 180,E1 -4329.139,E2 -4329.139} C_VEL
LIN {X 0,Y 531.034,Z 241.966,A -85,B 0,C 180,E1 -4332.226,E2 -4332.226} C_VEL
LIN {X 0,Y 530.99,Z 241.962,A -85,B 0,C 180,E1 -4335.351,E2 -4335.351} C_VEL
LIN {X 0,Y 530.987,Z 241.966,A -85,B 0,C 180,E1 -4338.522,E2 -4338.522} C_VEL
LIN {X 0,Y 530.994,Z 241.962,A -85,B 0,C 180,E1 -4340.939,E2 -4340.939} C_VEL
LIN {X 0,Y 530.975,Z 241.971,A -85,B 0,C 180,E1 -4344.225,E2 -4344.225} C_VEL
LIN {X 0,Y 531.002,Z 241.961,A -85,B 0,C 180,E1 -4346.745,E2 -4346.745} C_VEL
LIN {X 0,Y 530.989,Z 241.964,A -85,B 0,C 180,E1 -4349.323,E2 -4349.323} C_VEL
LIN {X 0,Y 530.977,Z 241.97,A -85,B 0,C 180,E1 -4352.104,E2 -4352.104} C_VEL
LIN {X 0,Y 530.985,Z 241.963,A -85,B 0,C 180,E1 -4354.855,E2 -4354.855} C_VEL
LIN {X 0,Y 530.964,Z 241.97,A -85,B 0,C 180,E1 -4357.509,E2 -4357.509} C_VEL
LIN {X 0,Y 530.981,Z 241.964,A -85,B 0,C 180,E1 -4360.434,E2 -4360.434} C_VEL
LIN {X 0,Y 530.961,Z 241.969,A -85,B 0,C 180,E1 -4363.282,E2 -4363.282} C_VEL
LIN {X 0,Y 530.987,Z 241.972,A -85,B 0,C 180,E1 -4365.622,E2 -4365.622} C_VEL
LIN {X 0,Y 530.996,Z 241.961,A -85,B 0,C 180,E1 -4368.566,E2 -4368.566} C_VEL
LIN {X 0,Y 530.956,Z 241.976,A -85,B 0,C 180,E1 -4371.53,E2 -4371.53} C_VEL
LIN {X 0,Y 530.954,Z 241.967,A -85,B 0,C 180,E1 -4374.381,E2 -4374.381} C_VEL
LIN {X 0,Y 530.971,Z 241.969,A -85,B 0,C 180,E1 -4377.134,E2 -4377.134} C_VEL
LIN {X 0,Y 530.97,Z 241.971,A -85,B 0,C 180,E1 -4379.804,E2 -4379.804} C_VEL
LIN {X 0,Y 531.014,Z 241.963,A -85,B 0,C 180,E1 -4382.468,E2 -4382.468} C_VEL
LIN {X 0,Y 531.036,Z 242.074,A -85,B 0,C 180,E1 -4384.265,E2 -4384.265} C_VEL
LIN {X 0,Y 532.874,Z 251.111,A -85,B 0,C 180,E1 -4385.676,E2 -4385.676} C_VEL
LIN {X 0,Y 532.627,Z 263.812,A -85,B 0,C 180,E1 -4387.502,E2 -4387.502} C_VEL
LIN {X 0,Y 532.06,Z 286.59,A -85,B 0,C 180,E1 -4390.718,E2 -4390.718} C_VEL
LIN {X 0,Y 531.938,Z 295.177,A -85,B 0,C 180,E1 -4391.885,E2 -4391.885} C_VEL
LIN {X 0,Y 533.899,Z 307.83,A -85,B 0,C 180,E1 -4392.129,E2 -4392.129} C_VEL
LIN {X 0,Y 533.267,Z 433.198,A -85,B 0,C 180,E1 -4393.86,E2 -4393.86} C_VEL
LIN {X 0,Y 533.023,Z 447.546,A -85,B 0,C 180,E1 -4394.214,E2 -4394.214} C_VEL
LIN {X 0,Y 532.778,Z 461.128,A -85,B 0,C 180,E1 -4394.703,E2 -4394.703} C_VEL
LIN {X 0,Y 532.449,Z 473.341,A -85,B 0,C 180,E1 -4395.281,E2 -4395.281} C_VEL
LIN {X 0,Y 532.088,Z 486.191,A -85,B 0,C 180,E1 -4396.052,E2 -4396.052} C_VEL
LIN {X 0,Y 531.749,Z 497.877,A -85,B 0,C 180,E1 -4396.919,E2 -4396.919} C_VEL
LIN {X 0,Y 531.459,Z 508.981,A -85,B 0,C 180,E1 -4397.921,E2 -4397.921} C_VEL
LIN {X 0,Y 531.204,Z 518.384,A -85,B 0,C 180,E1 -4398.94,E2 -4398.94} C_VEL
LIN {X 0,Y 530.921,Z 527.283,A -85,B 0,C 180,E1 -4400.091,E2 -4400.091} C_VEL
LIN {X 0,Y 530.736,Z 535.814,A -85,B 0,C 180,E1 -4401.433,E2 -4401.433} C_VEL
LIN {X 0,Y 530.587,Z 542.689,A -85,B 0,C 180,E1 -4402.771,E2 -4402.771} C_VEL
LIN {X 0,Y 530.565,Z 548.832,A -85,B 0,C 180,E1 -4404.298,E2 -4404.298} C_VEL
LIN {X 0,Y 530.447,Z 552.338,A -85,B 0,C 180,E1 -4405.44,E2 -4405.44} C_VEL
LIN {X 0,Y 530.453,Z 555.753,A -85,B 0,C 180,E1 -4406.962,E2 -4406.962} C_VEL
LIN {X 0,Y 530.357,Z 557.77,A -85,B 0,C 180,E1 -4408.481,E2 -4408.481} C_VEL
LIN {X 0,Y 530.341,Z 558.439,A -85,B 0,C 180,E1 -4410,E2 -4410} C_VEL
LIN {X 0,Y 530.357,Z 557.771,A -85,B 0,C 180,E1 -4411.519,E2 -4411.519} C_VEL
LIN {X 0,Y 530.453,Z 555.756,A -85,B 0,C 180,E1 -4413.038,E2 -4413.038} C_VEL
LIN {X 0,Y 530.447,Z 552.34,A -85,B 0,C 180,E1 -4414.559,E2 -4414.559} C_VEL
LIN {X 0,Y 530.547,Z 547.425,A -85,B 0,C 180,E1 -4416.083,E2 -4416.083} C_VEL
LIN {X 0,Y 530.641,Z 540.864,A -85,B 0,C 180,E1 -4417.611,E2 -4417.611} C_VEL
LIN {X 0,Y 530.789,Z 533.564,A -85,B 0,C 180,E1 -4418.95,E2 -4418.95} C_VEL
LIN {X 0,Y 531.011,Z 524.524,A -85,B 0,C 180,E1 -4420.292,E2 -4420.292} C_VEL
LIN {X 0,Y 531.29,Z 515.039,A -85,B 0,C 180,E1 -4421.444,E2 -4421.444} C_VEL
LIN {X 0,Y 531.555,Z 504.538,A -85,B 0,C 180,E1 -4422.503,E2 -4422.503} C_VEL
LIN {X 0,Y 531.87,Z 492.955,A -85,B 0,C 180,E1 -4423.467,E2 -4423.467} C_VEL
LIN {X 0,Y 532.267,Z 480.11,A -85,B 0,C 180,E1 -4424.334,E2 -4424.334} C_VEL
LIN {X 0,Y 532.579,Z 467.563,A -85,B 0,C 180,E1 -4425.009,E2 -4425.009} C_VEL
LIN {X 0,Y 532.923,Z 453.663,A -85,B 0,C 180,E1 -4425.584,E2 -4425.584} C_VEL
LIN {X 0,Y 533.179,Z 439.767,A -85,B 0,C 180,E1 -4425.998,E2 -4425.998} C_VEL
LIN {X 0,Y 533.301,Z 425.815,A -85,B 0,C 180,E1 -4426.262,E2 -4426.262} C_VEL
LIN {X 0,Y 533.812,Z 306.001,A -85,B 0,C 180,E1 -4427.899,E2 -4427.899} C_VEL
LIN {X 0,Y 531.891,Z 294.838,A -85,B 0,C 180,E1 -4428.123,E2 -4428.123} C_VEL
LIN {X 0,Y 532.367,Z 272.267,A -85,B 0,C 180,E1 -4431.286,E2 -4431.286} C_VEL
LIN {X 0,Y 532.864,Z 253.758,A -85,B 0,C 180,E1 -4433.926,E2 -4433.926} C_VEL
LIN {X 0,Y 532.517,Z 248.846,A -85,B 0,C 180,E1 -4434.657,E2 -4434.657} C_VEL
LIN {X 0,Y 531.019,Z 241.966,A -85,B 0,C 180,E1 -4435.761,E2 -4435.761} C_VEL
LIN {X 0,Y 530.997,Z 241.97,A -85,B 0,C 180,E1 -4438.455,E2 -4438.455} C_VEL
LIN {X 0,Y 530.958,Z 241.972,A -85,B 0,C 180,E1 -4441.078,E2 -4441.078} C_VEL
LIN {X 0,Y 530.987,Z 241.968,A -85,B 0,C 180,E1 -4443.772,E2 -4443.772} C_VEL
LIN {X 0,Y 530.953,Z 241.975,A -85,B 0,C 180,E1 -4446.558,E2 -4446.558} C_VEL
LIN {X 0,Y 530.984,Z 241.966,A -85,B 0,C 180,E1 -4449.442,E2 -4449.442} C_VEL
LIN {X 0,Y 530.98,Z 241.972,A -85,B 0,C 180,E1 -4452.455,E2 -4452.455} C_VEL
LIN {X 0,Y 530.983,Z 241.965,A -85,B 0,C 180,E1 -4455.62,E2 -4455.62} C_VEL
LIN {X 0,Y 530.997,Z 241.966,A -85,B 0,C 180,E1 -4458.564,E2 -4458.564} C_VEL
LIN {X 0,Y 530.955,Z 241.969,A -85,B 0,C 180,E1 -4461.528,E2 -4461.528} C_VEL
LIN {X 0,Y 530.978,Z 241.964,A -85,B 0,C 180,E1 -4464.381,E2 -4464.381} C_VEL
LIN {X 0,Y 530.967,Z 241.966,A -85,B 0,C 180,E1 -4467.133,E2 -4467.133} C_VEL
LIN {X 0,Y 530.981,Z 241.969,A -85,B 0,C 180,E1 -4469.803,E2 -4469.803} C_VEL
LIN {X 0,Y 531.011,Z 241.961,A -85,B 0,C 180,E1 -4472.466,E2 -4472.466} C_VEL
LIN {X 0,Y 530.999,Z 241.962,A -85,B 0,C 180,E1 -4474.941,E2 -4474.941} C_VEL
LIN {X 0,Y 530.964,Z 241.968,A -85,B 0,C 180,E1 -4478.246,E2 -4478.246} C_VEL
LIN {X 0,Y 530.989,Z 241.962,A -85,B 0,C 180,E1 -4480.676,E2 -4480.676} C_VEL
LIN {X 0,Y 530.986,Z 241.965,A -85,B 0,C 180,E1 -4483.07,E2 -4483.07} C_VEL
LIN {X 0,Y 531.011,Z 241.965,A -85,B 0,C 180,E1 -4485.435,E2 -4485.435} C_VEL
LIN {X 0,Y 531.038,Z 241.954,A -85,B 0,C 180,E1 -4488.549,E2 -4488.549} C_VEL
LIN {X 0,Y 531.052,Z 241.959,A -85,B 0,C 180,E1 -4491.628,E2 -4491.628} C_VEL
LIN {X 0,Y 531.116,Z 241.948,A -85,B 0,C 180,E1 -4494.684,E2 -4494.684} C_VEL
LIN {X 0,Y 531.128,Z 241.949,A -85,B 0,C 180,E1 -4497.724,E2 -4497.724} C_VEL
LIN {X 0,Y 531.147,Z 241.945,A -85,B 0,C 180,E1 -4500.757,E2 -4500.757} C_VEL
LIN {X 0,Y 531.1,Z 241.955,A -85,B 0,C 180,E1 -4503.033,E2 -4503.033} C_VEL
LIN {X 0,Y 531.073,Z 241.951,A -85,B 0,C 180,E1 -4506.076,E2 -4506.076} C_VEL
LIN {X 0,Y 531.022,Z 241.965,A -85,B 0,C 180,E1 -4509.137,E2 -4509.137} C_VEL
LIN {X 0,Y 531.029,Z 241.959,A -85,B 0,C 180,E1 -4512.224,E2 -4512.224} C_VEL
LIN {X 0,Y 530.984,Z 241.967,A -85,B 0,C 180,E1 -4515.349,E2 -4515.349} C_VEL
LIN {X 0,Y 530.978,Z 241.967,A -85,B 0,C 180,E1 -4518.52,E2 -4518.52} C_VEL
LIN {X 0,Y 530.992,Z 241.97,A -85,B 0,C 180,E1 -4520.937,E2 -4520.937} C_VEL
LIN {X 0,Y 530.994,Z 241.962,A -85,B 0,C 180,E1 -4524.044,E2 -4524.044} C_VEL
LIN {X 0,Y 530.991,Z 241.97,A -85,B 0,C 180,E1 -4526.743,E2 -4526.743} C_VEL
LIN {X 0,Y 530.986,Z 241.963,A -85,B 0,C 180,E1 -4529.321,E2 -4529.321} C_VEL
LIN {X 0,Y 530.955,Z 241.968,A -85,B 0,C 180,E1 -4532.101,E2 -4532.101} C_VEL
LIN {X 0,Y 530.97,Z 241.967,A -85,B 0,C 180,E1 -4534.853,E2 -4534.853} C_VEL
LIN {X 0,Y 530.951,Z 241.969,A -85,B 0,C 180,E1 -4537.507,E2 -4537.507} C_VEL
LIN {X 0,Y 531.011,Z 241.969,A -85,B 0,C 180,E1 -4540.428,E2 -4540.428} C_VEL
LIN {X 0,Y 530.949,Z 241.969,A -85,B 0,C 180,E1 -4543.579,E2 -4543.579} C_VEL
LIN {X 0,Y 530.276,Z 242.06,A -85,B 0,C 180,E1 -4544.213,E2 -4544.213} C_VEL
LIN {X 0,Y 527.427,Z 242.413,A -85,B 0,C 180,E1 -4545.242,E2 -4545.242} C_VEL
LIN {X 0,Y 525.024,Z 242.713,A -85,B 0,C 180,E1 -4546.07,E2 -4546.07} C_VEL
LIN {X 0,Y 523.991,Z 242.84,A -85,B 0,C 180,E1 -4546.71,E2 -4546.71} C_VEL
LIN {X 0,Y 523.906,Z 242.848,A -85,B 0,C 180,E1 -4546.926,E2 -4546.926} C_VEL
LIN {X 0,Y 523.963,Z 242.846,A -85,B 0,C 180,E1 -4549.923,E2 -4549.923} C_VEL
LIN {X 0,Y 523.975,Z 243.012,A -85,B 0,C 180,E1 -4553.407,E2 -4553.407} C_VEL
LIN {X 0,Y 525.307,Z 250.087,A -85,B 0,C 180,E1 -4554.694,E2 -4554.694} C_VEL
LIN {X 0,Y 524.894,Z 265.979,A -85,B 0,C 180,E1 -4557.384,E2 -4557.384} C_VEL
LIN {X 0,Y 524.868,Z 267.921,A -85,B 0,C 180,E1 -4557.691,E2 -4557.691} C_VEL
LIN {X 0,Y 527.159,Z 278.965,A -85,B 0,C 180,E1 -4557.931,E2 -4557.931} C_VEL
LIN {X 0,Y 526.502,Z 404.216,A -85,B 0,C 180,E1 -4559.685,E2 -4559.685} C_VEL
LIN {X 0,Y 526.225,Z 418.842,A -85,B 0,C 180,E1 -4560.048,E2 -4560.048} C_VEL
LIN {X 0,Y 525.973,Z 432.202,A -85,B 0,C 180,E1 -4560.536,E2 -4560.536} C_VEL
LIN {X 0,Y 525.628,Z 444.364,A -85,B 0,C 180,E1 -4561.118,E2 -4561.118} C_VEL
LIN {X 0,Y 525.267,Z 456.93,A -85,B 0,C 180,E1 -4561.882,E2 -4561.882} C_VEL
LIN {X 0,Y 524.874,Z 469.224,A -85,B 0,C 180,E1 -4562.812,E2 -4562.812} C_VEL
LIN {X 0,Y 524.531,Z 480.469,A -85,B 0,C 180,E1 -4563.855,E2 -4563.855} C_VEL
LIN {X 0,Y 524.183,Z 490.802,A -85,B 0,C 180,E1 -4565.018,E2 -4565.018} C_VEL
LIN {X 0,Y 523.931,Z 499.931,A -85,B 0,C 180,E1 -4566.271,E2 -4566.271} C_VEL
LIN {X 0,Y 523.699,Z 507.322,A -85,B 0,C 180,E1 -4567.503,E2 -4567.503} C_VEL
LIN {X 0,Y 523.549,Z 513.459,A -85,B 0,C 180,E1 -4568.75,E2 -4568.75} C_VEL
LIN {X 0,Y 523.476,Z 518.47,A -85,B 0,C 180,E1 -4570.012,E2 -4570.012} C_VEL
LIN {X 0,Y 523.384,Z 522.219,A -85,B 0,C 180,E1 -4571.2,E2 -4571.2} C_VEL
LIN {X 0,Y 523.313,Z 525.916,A -85,B 0,C 180,E1 -4572.816,E2 -4572.816} C_VEL
LIN {X 0,Y 523.252,Z 528.093,A -85,B 0,C 180,E1 -4574.418,E2 -4574.418} C_VEL
LIN {X 0,Y 523.321,Z 528.641,A -85,B 0,C 180,E1 -4575.217,E2 -4575.217} C_VEL
LIN {X 0,Y 523.266,Z 528.681,A -85,B 0,C 180,E1 -4576.802,E2 -4576.802} C_VEL
LIN {X 0,Y 523.319,Z 527.314,A -85,B 0,C 180,E1 -4578.379,E2 -4578.379} C_VEL
LIN {X 0,Y 523.321,Z 524.566,A -85,B 0,C 180,E1 -4579.946,E2 -4579.946} C_VEL
LIN {X 0,Y 523.419,Z 520.374,A -85,B 0,C 180,E1 -4581.507,E2 -4581.507} C_VEL
LIN {X 0,Y 523.533,Z 514.638,A -85,B 0,C 180,E1 -4583.061,E2 -4583.061} C_VEL
LIN {X 0,Y 523.624,Z 508.203,A -85,B 0,C 180,E1 -4584.416,E2 -4584.416} C_VEL
LIN {X 0,Y 523.885,Z 500.236,A -85,B 0,C 180,E1 -4585.769,E2 -4585.769} C_VEL
LIN {X 0,Y 524.119,Z 491.938,A -85,B 0,C 180,E1 -4586.926,E2 -4586.926} C_VEL
LIN {X 0,Y 524.456,Z 481.98,A -85,B 0,C 180,E1 -4588.08,E2 -4588.08} C_VEL
LIN {X 0,Y 524.814,Z 470.893,A -85,B 0,C 180,E1 -4589.137,E2 -4589.137} C_VEL
LIN {X 0,Y 525.242,Z 458.516,A -85,B 0,C 180,E1 -4590.096,E2 -4590.096} C_VEL
LIN {X 0,Y 525.631,Z 446.277,A -85,B 0,C 180,E1 -4590.862,E2 -4590.862} C_VEL
LIN {X 0,Y 525.954,Z 432.694,A -85,B 0,C 180,E1 -4591.531,E2 -4591.531} C_VEL
LIN {X 0,Y 526.247,Z 419.054,A -85,B 0,C 180,E1 -4592.033,E2 -4592.033} C_VEL
LIN {X 0,Y 526.422,Z 404.966,A -85,B 0,C 180,E1 -4592.391,E2 -4592.391} C_VEL
LIN {X 0,Y 526.985,Z 318.463,A -85,B 0,C 180,E1 -4593.608,E2 -4593.608} C_VEL
LIN {X 0,Y 527.13,Z 279.114,A -85,B 0,C 180,E1 -4594.157,E2 -4594.157} C_VEL
LIN {X 0,Y 524.856,Z 267.63,A -85,B 0,C 180,E1 -4594.416,E2 -4594.416} C_VEL
LIN {X 0,Y 525.196,Z 253.958,A -85,B 0,C 180,E1 -4596.724,E2 -4596.724} C_VEL
LIN {X 0,Y 525.198,Z 248.981,A -85,B 0,C 180,E1 -4597.575,E2 -4597.575} C_VEL
LIN {X 0,Y 524.014,Z 242.838,A -85,B 0,C 180,E1 -4598.727,E2 -4598.727} C_VEL
LIN {X 0,Y 524.01,Z 242.841,A -85,B 0,C 180,E1 -4601.751,E2 -4601.751} C_VEL
LIN {X 0,Y 523.978,Z 242.84,A -85,B 0,C 180,E1 -4605.053,E2 -4605.053} C_VEL
LIN {X 0,Y 523.95,Z 242.846,A -85,B 0,C 180,E1 -4607.969,E2 -4607.969} C_VEL
LIN {X 0,Y 523.958,Z 242.839,A -85,B 0,C 180,E1 -4610.41,E2 -4610.41} C_VEL
LIN {X 0,Y 523.931,Z 242.851,A -85,B 0,C 180,E1 -4613.729,E2 -4613.729} C_VEL
LIN {X 0,Y 523.967,Z 242.839,A -85,B 0,C 180,E1 -4616.271,E2 -4616.271} C_VEL
LIN {X 0,Y 523.956,Z 242.844,A -85,B 0,C 180,E1 -4619.327,E2 -4619.327} C_VEL
LIN {X 0,Y 523.927,Z 242.842,A -85,B 0,C 180,E1 -4622.449,E2 -4622.449} C_VEL
LIN {X 0,Y 523.922,Z 242.848,A -85,B 0,C 180,E1 -4625.226,E2 -4625.226} C_VEL
LIN {X 0,Y 523.904,Z 242.846,A -85,B 0,C 180,E1 -4628.102,E2 -4628.102} C_VEL
LIN {X 0,Y 523.956,Z 242.843,A -85,B 0,C 180,E1 -4631.09,E2 -4631.09} C_VEL
LIN {X 0,Y 523.928,Z 242.842,A -85,B 0,C 180,E1 -4634.228,E2 -4634.228} C_VEL
LIN {X 0,Y 523.913,Z 242.847,A -85,B 0,C 180,E1 -4636.834,E2 -4636.834} C_VEL
LIN {X 0,Y 523.955,Z 242.843,A -85,B 0,C 180,E1 -4638.911,E2 -4638.911} C_VEL
LIN {X 0,Y 523.904,Z 242.846,A -85,B 0,C 180,E1 -4641.899,E2 -4641.899} C_VEL
LIN {X 0,Y 523.927,Z 242.848,A -85,B 0,C 180,E1 -4644.909,E2 -4644.909} C_VEL
LIN {X 0,Y 523.93,Z 242.843,A -85,B 0,C 180,E1 -4647.679,E2 -4647.679} C_VEL
LIN {X 0,Y 523.957,Z 242.842,A -85,B 0,C 180,E1 -4650.674,E2 -4650.674} C_VEL
LIN {X 0,Y 523.966,Z 242.838,A -85,B 0,C 180,E1 -4653.73,E2 -4653.73} C_VEL
LIN {X 0,Y 523.924,Z 242.844,A -85,B 0,C 180,E1 -4656.272,E2 -4656.272} C_VEL
LIN {X 0,Y 523.936,Z 242.849,A -85,B 0,C 180,E1 -4658.768,E2 -4658.768} C_VEL
LIN {X 0,Y 523.943,Z 242.844,A -85,B 0,C 180,E1 -4661.222,E2 -4661.222} C_VEL
LIN {X 0,Y 523.93,Z 242.842,A -85,B 0,C 180,E1 -4663.64,E2 -4663.64} C_VEL
LIN {X 0,Y 523.931,Z 242.842,A -85,B 0,C 180,E1 -4666.029,E2 -4666.029} C_VEL
LIN {X 0,Y 524.001,Z 242.837,A -85,B 0,C 180,E1 -4668.395,E2 -4668.395} C_VEL
LIN {X 0,Y 523.996,Z 242.834,A -85,B 0,C 180,E1 -4671.517,E2 -4671.517} C_VEL
LIN {X 0,Y 524.089,Z 242.831,A -85,B 0,C 180,E1 -4674.615,E2 -4674.615} C_VEL
LIN {X 0,Y 524.103,Z 242.82,A -85,B 0,C 180,E1 -4677.696,E2 -4677.696} C_VEL
LIN {X 0,Y 524.117,Z 242.823,A -85,B 0,C 180,E1 -4680.769,E2 -4680.769} C_VEL
LIN {X 0,Y 524.067,Z 242.826,A -85,B 0,C 180,E1 -4683.076,E2 -4683.076} C_VEL
LIN {X 0,Y 524.039,Z 242.834,A -85,B 0,C 180,E1 -4686.16,E2 -4686.16} C_VEL
LIN {X 0,Y 523.993,Z 242.834,A -85,B 0,C 180,E1 -4689.263,E2 -4689.263} C_VEL
LIN {X 0,Y 523.995,Z 242.836,A -85,B 0,C 180,E1 -4691.74,E2 -4691.74} C_VEL
LIN {X 0,Y 523.986,Z 242.835,A -85,B 0,C 180,E1 -4695.053,E2 -4695.053} C_VEL
LIN {X 0,Y 523.959,Z 242.844,A -85,B 0,C 180,E1 -4697.97,E2 -4697.97} C_VEL
LIN {X 0,Y 523.966,Z 242.842,A -85,B 0,C 180,E1 -4700.411,E2 -4700.411} C_VEL
LIN {X 0,Y 523.912,Z 242.844,A -85,B 0,C 180,E1 -4702.894,E2 -4702.894} C_VEL
LIN {X 0,Y 523.948,Z 242.841,A -85,B 0,C 180,E1 -4705.42,E2 -4705.42} C_VEL
LIN {X 0,Y 523.966,Z 242.846,A -85,B 0,C 180,E1 -4708,E2 -4708} C_VEL
LIN {X 0,Y 523.949,Z 242.839,A -85,B 0,C 180,E1 -4710.857,E2 -4710.857} C_VEL
LIN {X 0,Y 523.958,Z 242.845,A -85,B 0,C 180,E1 -4713.736,E2 -4713.736} C_VEL
LIN {X 0,Y 523.92,Z 242.845,A -85,B 0,C 180,E1 -4716.405,E2 -4716.405} C_VEL
LIN {X 0,Y 523.92,Z 242.844,A -85,B 0,C 180,E1 -4719.086,E2 -4719.086} C_VEL
LIN {X 0,Y 523.951,Z 242.843,A -85,B 0,C 180,E1 -4722.12,E2 -4722.12} C_VEL
LIN {X 0,Y 523.955,Z 242.843,A -85,B 0,C 180,E1 -4725.31,E2 -4725.31} C_VEL
LIN {X 0,Y 523.958,Z 242.838,A -85,B 0,C 180,E1 -4728.69,E2 -4728.69} C_VEL
LIN {X 0,Y 523.916,Z 242.846,A -85,B 0,C 180,E1 -4731.081,E2 -4731.081} C_VEL
LIN {X 0,Y 523.9,Z 242.85,A -85,B 0,C 180,E1 -4733.826,E2 -4733.826} C_VEL
LIN {X 0,Y 523.942,Z 242.841,A -85,B 0,C 180,E1 -4736.636,E2 -4736.636} C_VEL
LIN {X 0,Y 523.957,Z 242.849,A -85,B 0,C 180,E1 -4739.356,E2 -4739.356} C_VEL
LIN {X 0,Y 523.978,Z 242.84,A -85,B 0,C 180,E1 -4742.282,E2 -4742.282} C_VEL
LIN {X 0,Y 524.01,Z 243.029,A -85,B 0,C 180,E1 -4744.066,E2 -4744.066} C_VEL
LIN {X 0,Y 525.964,Z 252.253,A -85,B 0,C 180,E1 -4745.53,E2 -4745.53} C_VEL
LIN {X 0,Y 525.748,Z 264.218,A -85,B 0,C 180,E1 -4747.275,E2 -4747.275} C_VEL
LIN {X 0,Y 525.102,Z 286.389,A -85,B 0,C 180,E1 -4750.452,E2 -4750.452} C_VEL
LIN {X 0,Y 524.936,Z 294.71,A -85,B 0,C 180,E1 -4751.631,E2 -4751.631} C_VEL
LIN {X 0,Y 527.135,Z 307.875,A -85,B 0,C 180,E1 -4751.895,E2 -4751.895} C_VEL
LIN {X 0,Y 526.45,Z 432.956,A -85,B 0,C 180,E1 -4753.645,E2 -4753.645} C_VEL
LIN {X 0,Y 526.19,Z 446.958,A -85,B 0,C 180,E1 -4753.991,E2 -4753.991} C_VEL
LIN {X 0,Y 525.913,Z 460.908,A -85,B 0,C 180,E1 -4754.498,E2 -4754.498} C_VEL
LIN {X 0,Y 525.555,Z 473.125,A -85,B 0,C 180,E1 -4755.083,E2 -4755.083} C_VEL
LIN {X 0,Y 525.168,Z 485.979,A -85,B 0,C 180,E1 -4755.864,E2 -4755.864} C_VEL
LIN {X 0,Y 524.801,Z 497.668,A -85,B 0,C 180,E1 -4756.742,E2 -4756.742} C_VEL
LIN {X 0,Y 524.449,Z 509.122,A -85,B 0,C 180,E1 -4757.792,E2 -4757.792} C_VEL
LIN {X 0,Y 524.145,Z 519.814,A -85,B 0,C 180,E1 -4758.985,E2 -4758.985} C_VEL
LIN {X 0,Y 523.845,Z 528.441,A -85,B 0,C 180,E1 -4760.151,E2 -4760.151} C_VEL
LIN {X 0,Y 523.67,Z 536.706,A -85,B 0,C 180,E1 -4761.511,E2 -4761.511} C_VEL
LIN {X 0,Y 523.503,Z 542.488,A -85,B 0,C 180,E1 -4762.673,E2 -4762.673} C_VEL
LIN {X 0,Y 523.453,Z 547.229,A -85,B 0,C 180,E1 -4763.834,E2 -4763.834} C_VEL
LIN {X 0,Y 523.377,Z 551.067,A -85,B 0,C 180,E1 -4764.993,E2 -4764.993} C_VEL
LIN {X 0,Y 523.419,Z 554.027,A -85,B 0,C 180,E1 -4766.151,E2 -4766.151} C_VEL
LIN {X 0,Y 523.334,Z 556.733,A -85,B 0,C 180,E1 -4767.691,E2 -4767.691} C_VEL
LIN {X 0,Y 523.248,Z 558.073,A -85,B 0,C 180,E1 -4769.23,E2 -4769.23} C_VEL
LIN {X 0,Y 523.248,Z 558.072,A -85,B 0,C 180,E1 -4770.769,E2 -4770.769} C_VEL
LIN {X 0,Y 523.334,Z 556.734,A -85,B 0,C 180,E1 -4772.309,E2 -4772.309} C_VEL
LIN {X 0,Y 523.419,Z 554.028,A -85,B 0,C 180,E1 -4773.849,E2 -4773.849} C_VEL
LIN {X 0,Y 523.449,Z 549.875,A -85,B 0,C 180,E1 -4775.393,E2 -4775.393} C_VEL
LIN {X 0,Y 523.495,Z 544.155,A -85,B 0,C 180,E1 -4776.94,E2 -4776.94} C_VEL
LIN {X 0,Y 523.635,Z 537.709,A -85,B 0,C 180,E1 -4778.295,E2 -4778.295} C_VEL
LIN {X 0,Y 523.834,Z 529.7,A -85,B 0,C 180,E1 -4779.654,E2 -4779.654} C_VEL
LIN {X 0,Y 524.091,Z 521.325,A -85,B 0,C 180,E1 -4780.82,E2 -4780.82} C_VEL
LIN {X 0,Y 524.391,Z 510.613,A -85,B 0,C 180,E1 -4782.057,E2 -4782.057} C_VEL
LIN {X 0,Y 524.721,Z 499.996,A -85,B 0,C 180,E1 -4783.062,E2 -4783.062} C_VEL
LIN {X 0,Y 525.061,Z 488.811,A -85,B 0,C 180,E1 -4783.941,E2 -4783.941} C_VEL
LIN {X 0,Y 525.437,Z 476.632,A -85,B 0,C 180,E1 -4784.722,E2 -4784.722} C_VEL
LIN {X 0,Y 525.828,Z 463.121,A -85,B 0,C 180,E1 -4785.405,E2 -4785.405} C_VEL
LIN {X 0,Y 526.125,Z 448.998,A -85,B 0,C 180,E1 -4785.942,E2 -4785.942} C_VEL
LIN {X 0,Y 526.397,Z 435.186,A -85,B 0,C 180,E1 -4786.307,E2 -4786.307} C_VEL
LIN {X 0,Y 526.545,Z 413.025,A -85,B 0,C 180,E1 -4786.651,E2 -4786.651} C_VEL
LIN {X 0,Y 527.05,Z 306.939,A -85,B 0,C 180,E1 -4788.12,E2 -4788.12} C_VEL
LIN {X 0,Y 524.927,Z 294.549,A -85,B 0,C 180,E1 -4788.383,E2 -4788.383} C_VEL
LIN {X 0,Y 525.49,Z 272.082,A -85,B 0,C 180,E1 -4791.579,E2 -4791.579} C_VEL
LIN {X 0,Y 526.017,Z 253.598,A -85,B 0,C 180,E1 -4794.257,E2 -4794.257} C_VEL
LIN {X 0,Y 524.764,Z 246.462,A -85,B 0,C 180,E1 -4795.376,E2 -4795.376} C_VEL
LIN {X 0,Y 523.963,Z 242.846,A -85,B 0,C 180,E1 -4795.978,E2 -4795.978} C_VEL
LIN {X 0,Y 523.939,Z 242.847,A -85,B 0,C 180,E1 -4798.874,E2 -4798.874} C_VEL
LIN {X 0,Y 523.923,Z 242.847,A -85,B 0,C 180,E1 -4801.543,E2 -4801.543} C_VEL
LIN {X 0,Y 523.932,Z 242.852,A -85,B 0,C 180,E1 -4804.289,E2 -4804.289} C_VEL
LIN {X 0,Y 523.905,Z 242.847,A -85,B 0,C 180,E1 -4807.131,E2 -4807.131} C_VEL
LIN {X 0,Y 523.936,Z 242.85,A -85,B 0,C 180,E1 -4810.129,E2 -4810.129} C_VEL
LIN {X 0,Y 523.937,Z 242.849,A -85,B 0,C 180,E1 -4812.458,E2 -4812.458} C_VEL
LIN {X 0,Y 523.952,Z 242.84,A -85,B 0,C 180,E1 -4815.308,E2 -4815.308} C_VEL
LIN {X 0,Y 523.958,Z 242.842,A -85,B 0,C 180,E1 -4818.688,E2 -4818.688} C_VEL
LIN {X 0,Y 523.913,Z 242.851,A -85,B 0,C 180,E1 -4821.897,E2 -4821.897} C_VEL
LIN {X 0,Y 523.934,Z 242.837,A -85,B 0,C 180,E1 -4824.908,E2 -4824.908} C_VEL
LIN {X 0,Y 523.938,Z 242.846,A -85,B 0,C 180,E1 -4827.677,E2 -4827.677} C_VEL
LIN {X 0,Y 523.957,Z 242.84,A -85,B 0,C 180,E1 -4830.674,E2 -4830.674} C_VEL
LIN {X 0,Y 523.969,Z 242.844,A -85,B 0,C 180,E1 -4833.727,E2 -4833.727} C_VEL
LIN {X 0,Y 523.93,Z 242.844,A -85,B 0,C 180,E1 -4836.27,E2 -4836.27} C_VEL
LIN {X 0,Y 523.939,Z 242.841,A -85,B 0,C 180,E1 -4838.766,E2 -4838.766} C_VEL
LIN {X 0,Y 523.946,Z 242.842,A -85,B 0,C 180,E1 -4841.22,E2 -4841.22} C_VEL
LIN {X 0,Y 523.934,Z 242.847,A -85,B 0,C 180,E1 -4843.638,E2 -4843.638} C_VEL
LIN {X 0,Y 523.933,Z 242.845,A -85,B 0,C 180,E1 -4846.027,E2 -4846.027} C_VEL
LIN {X 0,Y 524.003,Z 242.831,A -85,B 0,C 180,E1 -4848.393,E2 -4848.393} C_VEL
LIN {X 0,Y 523.999,Z 242.839,A -85,B 0,C 180,E1 -4851.515,E2 -4851.515} C_VEL
LIN {X 0,Y 524.077,Z 242.825,A -85,B 0,C 180,E1 -4854.613,E2 -4854.613} C_VEL
LIN {X 0,Y 524.101,Z 242.825,A -85,B 0,C 180,E1 -4857.693,E2 -4857.693} C_VEL
LIN {X 0,Y 524.116,Z 242.821,A -85,B 0,C 180,E1 -4860.767,E2 -4860.767} C_VEL
LIN {X 0,Y 524.066,Z 242.831,A -85,B 0,C 180,E1 -4863.074,E2 -4863.074} C_VEL
LIN {X 0,Y 524.035,Z 242.828,A -85,B 0,C 180,E1 -4866.158,E2 -4866.158} C_VEL
